{attribute 'global_init_slot' := '40510'}
VAR_GLOBAL
  LblAggregates_FunctionallyIndependentEequipment                 :FB_BA_Label:=( sObjName:='FIE',sDescr:='Functionally independent equipment');
  LblAggregates_SelfContainedControlUnit                          :FB_BA_Label:=( sObjName:='SCR',sDescr:='Self-contained control or regulation unit');
  LblAggregates_ControlCabinet                                    :FB_BA_Label:=( sObjName:='CCB',sDescr:='Control cabinet (trade-specific)');
//330 Doors, gates, windows, sun protection
  LblAggregates_WindowDrive                                       :FB_BA_Label:=( sObjName:='WIN',sDescr:='Window (drive)');
  LblAggregates_WindowContact                                     :FB_BA_Label:=( sObjName:='WIC',sDescr:='Window contact');
  LblAggregates_Blind                                             :FB_BA_Label:=( sObjName:='BLD',sDescr:='Blind');
  LblAggregates_Awning                                            :FB_BA_Label:=( sObjName:='AWN',sDescr:='Awning');
  LblAggregates_RollerShutters                                    :FB_BA_Label:=( sObjName:='ROS',sDescr:='Roller shutters');
  LblAggregates_Gate                                              :FB_BA_Label:=( sObjName:='GAT',sDescr:='Gate');
  LblAggregates_Door                                              :FB_BA_Label:=( sObjName:='DOR',sDescr:='Door');
  LblAggregates_DoorContact                                       :FB_BA_Label:=( sObjName:='DOC',sDescr:='Door contact');
  LblAggregates_Blackout                                          :FB_BA_Label:=( sObjName:='BLA',sDescr:='Blackout');
//412 Water plants
  LblAggregates_TraceHeating                                      :FB_BA_Label:=( sObjName:='THT',sDescr:='Trace heating');
  LblAggregates_ElectricHeating                                   :FB_BA_Label:=( sObjName:='EHT',sDescr:='Electric heating (warm water temperature preparation)');
  LblAggregates_WaterFilter                                       :FB_BA_Label:=( sObjName:='WFL',sDescr:='Water filter');
//421 Heat generation plants
  LblAggregates_Furnace                                           :FB_BA_Label:=( sObjName:='FUR',sDescr:='Furnace');
  LblAggregates_HeatExchanger                                     :FB_BA_Label:=( sObjName:='HEX',sDescr:='Heat exchanger');
//430 Ventilation and refrigeration systems
  LblAggregates_FanExhaustAir                                     :FB_BA_Label:=( sObjName:='EHF',sDescr:='Exhaust air fan');
  LblAggregates_Airwasher                                         :FB_BA_Label:=( sObjName:='AWA',sDescr:='Airwasher');
  LblAggregates_Humidifier                                        :FB_BA_Label:=( sObjName:='HUF',sDescr:='Humidifier');
  LblAggregates_HumidifierPump                                    :FB_BA_Label:=( sObjName:='HUP',sDescr:='Humidifier pump');
  LblAggregates_FireDamper                                        :FB_BA_Label:=( sObjName:='FID',sDescr:='Fire damper, fire protection valve');
  LblAggregates_SmokeProtectionDamper                             :FB_BA_Label:=( sObjName:='SPD',sDescr:='Smoke protection damper');
  LblAggregates_SmokeExtractorDamper                              :FB_BA_Label:=( sObjName:='SEP',sDescr:='Smoke extractor damper');
  LblAggregates_CeilingSwirlDiffuser                              :FB_BA_Label:=( sObjName:='CSD',sDescr:='Ceiling swirl diffuser');
  LblAggregates_RoofAirHeater                                     :FB_BA_Label:=( sObjName:='RAH',sDescr:='Roof air heater');
  LblAggregates_DirectEvaporator                                  :FB_BA_Label:=( sObjName:='DEA',sDescr:='Direct evaporator');
  LblAggregates_ElectricalAirHeater                               :FB_BA_Label:=( sObjName:='EAH',sDescr:='Electrical air heater');
  LblAggregates_ElectricReHeater                                  :FB_BA_Label:=( sObjName:='ERH',sDescr:='Electric re-heater');
  LblAggregates_ElectricaPreHeater                                :FB_BA_Label:=( sObjName:='EPH',sDescr:='Electrical pre-heater');
  LblAggregates_HeaterGeneral                                     :FB_BA_Label:=( sObjName:='HTR',sDescr:='Heater ');
  LblAggregates_FanExtractAir                                     :FB_BA_Label:=( sObjName:='EXF',sDescr:='Extract air fan ');
  LblAggregates_InductionDevice                                   :FB_BA_Label:=( sObjName:='IND',sDescr:='Induction device');
  LblAggregates_RefrigerantDryer                                  :FB_BA_Label:=( sObjName:='RFD',sDescr:='Refrigerant dryer');
  LblAggregates_CirculatorySystem                                 :FB_BA_Label:=( sObjName:='CCS',sDescr:='Circulatory system ');
  LblAggregates_AirFilterOutsideAir                               :FB_BA_Label:=( sObjName:='AFI',sDescr:='Outside air filter');
  LblAggregates_AirFilterSupplyAir                                :FB_BA_Label:=( sObjName:='AFI',sDescr:='Supply air filter');
  LblAggregates_AirFilterExhaustAir                               :FB_BA_Label:=( sObjName:='AFI',sDescr:='Exhaus air filter');
  LblAggregates_AirFilterExtractAir                               :FB_BA_Label:=( sObjName:='AFI',sDescr:='Extract air filter');
  LblAggregates_AirFilter                                         :FB_BA_Label:=( sObjName:='AFI',sDescr:='Air filter');
  LblAggregates_VentilationDamper                                 :FB_BA_Label:=( sObjName:='VFL',sDescr:='Ventilation flap');
  LblAggregates_VentilationDamperOutsideAir                       :FB_BA_Label:=( sObjName:='VFL',sDescr:='Ventilation flap outside air');
  LblAggregates_VentilationDamperExhaustAir                       :FB_BA_Label:=( sObjName:='VFL',sDescr:='Ventilation flap exhaust air');
  LblAggregates_VentilationDamperMixAir                           :FB_BA_Label:=( sObjName:='VFL',sDescr:='Ventilation flap mix air');
  LblAggregates_VentilationDamperSupplyAir                        :FB_BA_Label:=( sObjName:='VFL',sDescr:='Ventilation flap supply air');
  LblAggregates_VentilationDamperBypassAir                        :FB_BA_Label:=( sObjName:='VFL',sDescr:='Ventilation flap bypass');
  LblAggregates_Pump                                              :FB_BA_Label:=( sObjName:='PUM',sDescr:='Pump');
  LblAggregates_RecirculatingAirCoolingDevice                     :FB_BA_Label:=( sObjName:='RAC',sDescr:='Recirculating air cooling device');
  LblAggregates_FanRecirculatingAir                               :FB_BA_Label:=( sObjName:='RAF',sDescr:='Recirculating air fan');
  LblAggregates_UvFilter                                          :FB_BA_Label:=( sObjName:='UVF',sDescr:='UV filter');
  LblAggregates_VariableFlowRateController                        :FB_BA_Label:=( sObjName:='VFC',sDescr:='Variable flow rate controller');
  LblAggregates_WaterAirHeater                                    :FB_BA_Label:=( sObjName:='WAH',sDescr:='Water air heater');
  LblAggregates_WaterReHeater                                     :FB_BA_Label:=( sObjName:='WRH',sDescr:='Water re-heater');
  LblAggregates_WaterPreHeater                                    :FB_BA_Label:=( sObjName:='WPH',sDescr:='Water pre-heater');
  LblAggregates_HeatRecovery                                      :FB_BA_Label:=( sObjName:='HRC',sDescr:='Heat recovery');
  LblAggregates_FanSupplyAir                                      :FB_BA_Label:=( sObjName:='SUF',sDescr:='Supply air fan');
  LblAggregates_SmokeExtractionSystems                            :FB_BA_Label:=( sObjName:='SES',sDescr:='Smoke extraction systems');
  LblAggregates_SmokeExtractionVentilator                         :FB_BA_Label:=( sObjName:='SEF',sDescr:='Smoke extraction fan');
  LblAggregates_VentWindow                                        :FB_BA_Label:=( sObjName:='VWI',sDescr:='Vent window');
  LblAggregates_VentFlap                                          :FB_BA_Label:=( sObjName:='VFL',sDescr:='Vent flap');
  LblAggregates_VentDoor                                          :FB_BA_Label:=( sObjName:='VDO',sDescr:='Vent door');
  LblAggregates_WakeFan                                           :FB_BA_Label:=( sObjName:='WAF',sDescr:='Wake fan');
//434 Refrigeration systems
  LblAggregates_GlycoOilProtector                                 :FB_BA_Label:=( sObjName:='GLP',sDescr:='Glycol/oil protector');
  LblAggregates_Chiller                                           :FB_BA_Label:=( sObjName:='CHI',sDescr:='Chiller');
  LblAggregates_ReCoolingPlant                                    :FB_BA_Label:=( sObjName:='RCP',sDescr:='Re-cooling plant');
//440 High-voltage systems
  LblAggregates_GeneralPowerSupply                                :FB_BA_Label:=( sObjName:='GPS',sDescr:='General power supply');
  LblAggregates_CombindeHeatPowerStation                          :FB_BA_Label:=( sObjName:='CGU',sDescr:='Co-generation unit');
  LblAggregates_CompensationSystem                                :FB_BA_Label:=( sObjName:='CPS',sDescr:='Compensation system');
  LblAggregates_CouplingSwitch                                    :FB_BA_Label:=( sObjName:='COS',sDescr:='Coupling switch');
  LblAggregates_LoadBreakSwitch                                   :FB_BA_Label:=( sObjName:='LBS',sDescr:='Load-break switch');
  LblAggregates_CircuitBreaker                                    :FB_BA_Label:=( sObjName:='CCB',sDescr:='Circuit breaker');
  LblAggregates_NetworkAnalyser                                   :FB_BA_Label:=( sObjName:='NWA',sDescr:='Network analyser');
  LblAggregates_EmergencyPoweGeneratorUnit                        :FB_BA_Label:=( sObjName:='EPG',sDescr:='Emergency power generator unit');
  LblAggregates_EmergencyLighting                                 :FB_BA_Label:=( sObjName:='EML',sDescr:='Emergency lighting');
  LblAggregates_SafetyPowerSupply                                 :FB_BA_Label:=( sObjName:='SPS',sDescr:='Safety power supply');
  LblAggregates_Transformer                                       :FB_BA_Label:=( sObjName:='TRF',sDescr:='Transformer');
  LblAggregates_UninterruptiblePowerSupply                        :FB_BA_Label:=( sObjName:='UPS',sDescr:='Uninterruptible power supply');
//450 Telecommunications and information technology equipment
  LblAggregates_CentralFireAlarmSystem                            :FB_BA_Label:=( sObjName:='CFA',sDescr:='Central fire alarm system');
  LblAggregates_FireControlPanel                                  :FB_BA_Label:=( sObjName:='FCP',sDescr:='Fire control panel');
  LblAggregates_KitchenTableau                                    :FB_BA_Label:=( sObjName:='KIT',sDescr:='Kitchen tableau');
  LblAggregates_SmokeDetector                                     :FB_BA_Label:=( sObjName:='SDE',sDescr:='Smoke detector');
  LblAggregates_SmokeProtectionScreen                             :FB_BA_Label:=( sObjName:='SPS',sDescr:='Smoke protection screen');
  LblAggregates_VoiceAlarmCentre                                  :FB_BA_Label:=( sObjName:='VAC',sDescr:='Voice alarm centre');
  LblAggregates_Tableau                                           :FB_BA_Label:=( sObjName:='TAB',sDescr:='Tableau (general)');
//460 Conveyors
  LblAggregates_LiftGeneral                                       :FB_BA_Label:=( sObjName:='LIG',sDescr:='Lift general');
  LblAggregates_GoodsLift                                         :FB_BA_Label:=( sObjName:='GLI',sDescr:='Goods lift');
  LblAggregates_PassengerLift                                     :FB_BA_Label:=( sObjName:='PLI',sDescr:='Passenger lift');
//470 User-specific systems
  LblAggregates_FumeCupboard                                      :FB_BA_Label:=( sObjName:='FCB',sDescr:='Fume cupboard');
  LblAggregates_Compressor                                        :FB_BA_Label:=( sObjName:='COM',sDescr:='Compressor');
  LblAggregates_ProgrammableLogicControllers                      :FB_BA_Label:=( sObjName:='PLC',sDescr:='Programmable logic controllers');
//479 User-specific system, weather station
  LblAggregates_RainSensor                                        :FB_BA_Label:=( sObjName:='RAS',sDescr:='Rain sensor');
  LblAggregates_SolarRadiation                                    :FB_BA_Label:=( sObjName:='SOR',sDescr:='Solar radiation');
  LblAggregates_WeatherStation                                    :FB_BA_Label:=( sObjName:='WST',sDescr:='Weather station');
  LblAggregates_WindSpeed                                         :FB_BA_Label:=( sObjName:='WIS',sDescr:='Wind speed');
  LblAggregates_WindDirection                                     :FB_BA_Label:=( sObjName:='WID',sDescr:='Wind direction');
  LblAggregates_WindForce                                         :FB_BA_Label:=( sObjName:='WDF',sDescr:='Wind force');
  LblAggregates_Brightness                                        :FB_BA_Label:=( sObjName:='BIN',sDescr:='Brightness');
  LblAggregates_Dawn                                              :FB_BA_Label:=( sObjName:='BID',sDescr:='Brightness dawn');
  LblAggregates_PressureAbsolute                                  :FB_BA_Label:=( sObjName:='PAB',sDescr:='Pressure absolute');
  LblAggregates_PressureRelative                                  :FB_BA_Label:=( sObjName:='PRE',sDescr:='Pressure relative');
  LblAggregates_GeoLatitude                                       :FB_BA_Label:=( sObjName:='LAT',sDescr:='Latitude       ');
  LblAggregates_GeoLongitude                                      :FB_BA_Label:=( sObjName:='LOT',sDescr:='Longitude      ');
  LblAggregates_SunAzimuth                                        :FB_BA_Label:=( sObjName:='AZI',sDescr:='Azimuth        ');
  LblAggregates_SunElevation                                      :FB_BA_Label:=( sObjName:='ELE',sDescr:='Elevation      ');
//480 Building automation and control systems
  LblAggregates_SystemSwitch                                      :FB_BA_Label:=( sObjName:='SYS',sDescr:='System switch');
  LblAggregates_AutomationStationEquipment                        :FB_BA_Label:=( sObjName:='ASE',sDescr:='Automation station equipment');
  LblAggregates_BusLineCoupler                                    :FB_BA_Label:=( sObjName:='BUS',sDescr:='Bus line coupler');
  LblAggregates_DataInterfaceUnit                                 :FB_BA_Label:=( sObjName:='DIU',sDescr:='Data interface unit');
  LblAggregates_FieldbusModule                                    :FB_BA_Label:=( sObjName:='FBM',sDescr:='Fieldbus module');
  LblAggregates_InformationFocalPoint                             :FB_BA_Label:=( sObjName:='IFP',sDescr:='Information focal point');
  LblAggregates_ManagementAndControlEquipment                     :FB_BA_Label:=( sObjName:='MCE',sDescr:='Management and control equipment');
//481 BACS sensors – temperature
  LblAggregates_TemperatureGasEmission                            :FB_BA_Label:=( sObjName:='TEG',sDescr:='Emissions gas temperature');
  LblAggregates_TemperatureExtractAir                             :FB_BA_Label:=( sObjName:='TEX',sDescr:='Extract air temperature');
  LblAggregates_TemperatureOutside                                :FB_BA_Label:=( sObjName:='TOU',sDescr:='Outside temperature');
  LblAggregates_TemperatureExhaustAir                             :FB_BA_Label:=( sObjName:='TEH',sDescr:='Exhaust air temperature');
  LblAggregates_FrostProtectionMonitor                            :FB_BA_Label:=( sObjName:='FPM',sDescr:='Frost protection monitor');
  LblAggregates_TemperatureMixedAir                               :FB_BA_Label:=( sObjName:='TMI',sDescr:='Mixed air temperature');
  LblAggregates_TemperatureRoomAir                                :FB_BA_Label:=( sObjName:='TRO',sDescr:='Room temperature');
  LblAggregates_TemperatureReturnFlow                             :FB_BA_Label:=( sObjName:='TRT',sDescr:='Return flow temperature');
  LblAggregates_LimiterSafetyTemperature                          :FB_BA_Label:=( sObjName:='STL',sDescr:='Safety temperature limiter');
  LblAggregates_MonitorSafetyTemperature                          :FB_BA_Label:=( sObjName:='STM',sDescr:='Safety temperature monitor');
  LblAggregates_TemperatureStorage                                :FB_BA_Label:=( sObjName:='TST',sDescr:='Storage temperature');
  LblAggregates_TemperatureDewPoint                               :FB_BA_Label:=( sObjName:='TDP',sDescr:='Dew point temperature');
  LblAggregates_MonitorDewPoint                                   :FB_BA_Label:=( sObjName:='DPM',sDescr:='Dew point monitor');
  LblAggregates_TemperatureAfterCooler                            :FB_BA_Label:=( sObjName:='TAC',sDescr:='Temperature after cooler');
  LblAggregates_TemperatureAfterPreHeater                         :FB_BA_Label:=( sObjName:='TAP',sDescr:='Temperature after pre-heater');
  LblAggregates_TemperatureAfterHeatRecovery                      :FB_BA_Label:=( sObjName:='TAR',sDescr:='Temperature after heat recovery');
  LblAggregates_Thermostat                                        :FB_BA_Label:=( sObjName:='THM',sDescr:='Thermostat');
  LblAggregates_TemperatureHotWater                               :FB_BA_Label:=( sObjName:='THW',sDescr:='Hot water temperature');
  LblAggregates_TemperatureCirculation                            :FB_BA_Label:=( sObjName:='TCI',sDescr:='Circulation temperature');
  LblAggregates_TemperatureRecirculatingAir                       :FB_BA_Label:=( sObjName:='TRE',sDescr:='Recirculating air temperature');
  LblAggregates_TemperatureFlow                                   :FB_BA_Label:=( sObjName:='TFL',sDescr:='Flow temperature');
  LblAggregates_TemperatureSupplyAir                              :FB_BA_Label:=( sObjName:='TSU',sDescr:='Supply air temperature');
//481 BACS sensors – pressure
  LblAggregates_PressureExtractAir                                :FB_BA_Label:=( sObjName:='PEX',sDescr:='Extract air pressure');
  LblAggregates_PressureOutsideAir                                :FB_BA_Label:=( sObjName:='POU',sDescr:='Outside air pressure');
  LblAggregates_PressureDifferential                              :FB_BA_Label:=( sObjName:='PDI',sDescr:='Differential pressure');
  LblAggregates_PressureDifferentialOutsideAirFilter              :FB_BA_Label:=( sObjName:='PDI',sDescr:='Differential pressure outside air filter');
  LblAggregates_PressureDifferentialExtractAirFilter              :FB_BA_Label:=( sObjName:='PDI',sDescr:='Differential pressure extract air filter');
  LblAggregates_PressureDifferentialExhaustAirFilter              :FB_BA_Label:=( sObjName:='PDI',sDescr:='Differential pressure exhaust air filter');
  LblAggregates_PressureDifferentialSupplyAirFan                  :FB_BA_Label:=( sObjName:='PDI',sDescr:='Differential pressure supply air fan');
  LblAggregates_PressureDifferentialExtractAirFan                 :FB_BA_Label:=( sObjName:='PDI',sDescr:='Differential pressure ectract air fan');
  LblAggregates_PressureDifferentialExhaustAirFan                 :FB_BA_Label:=( sObjName:='PDI',sDescr:='Differential pressure exhaust air fan');
  LblAggregates_PressureSensorFlow                                :FB_BA_Label:=( sObjName:='PFL',sDescr:='Pressure sensor (water) flow');
  LblAggregates_MonitorPressure                                   :FB_BA_Label:=( sObjName:='PCO',sDescr:='Pressure controller');
  LblAggregates_PressureExhaustAir                                :FB_BA_Label:=( sObjName:='PEH',sDescr:='Exhaust air pressure');
  LblAggregates_PressureRoomAir                                   :FB_BA_Label:=( sObjName:='PRO',sDescr:='Room pressure');
  LblAggregates_PressureIndexCircuitSensorDifferential            :FB_BA_Label:=( sObjName:='PSI',sDescr:='Index circuit sensor differential pressure');
  LblAggregates_LimiterSafetyPressure                             :FB_BA_Label:=( sObjName:='SPL',sDescr:='Safety pressure limiter');
  LblAggregates_PressureSupplyAir                                 :FB_BA_Label:=( sObjName:='PSU',sDescr:='Supply air pressure');
//481 BACS sensors – air quality
  LblAggregates_CO2Sensor                                         :FB_BA_Label:=( sObjName:='COM',sDescr:='CO2 sensor');
  LblAggregates_QualityExtractAir                                 :FB_BA_Label:=( sObjName:='QEX',sDescr:='Extract air quality');
  LblAggregates_OualityRoomAir                                    :FB_BA_Label:=( sObjName:='QRO',sDescr:='Room air quality');
  LblAggregates_QualitiySupplyAir                                 :FB_BA_Label:=( sObjName:='QSU',sDescr:='Supply air quality');
  LblAggregates_QualityAirSensor                                  :FB_BA_Label:=( sObjName:='AQS',sDescr:='Air quality sensor');
//481 BACS sensors – humidity
  LblAggregates_Hygrostat                                         :FB_BA_Label:=( sObjName:='HYG',sDescr:='Hygrostat');
  LblAggregates_RelativeHumiditiyExtractAir                       :FB_BA_Label:=( sObjName:='HEX',sDescr:='Relative extract air humidity');
  LblAggregates_RelativeHumidityOutsideAir                        :FB_BA_Label:=( sObjName:='HOU',sDescr:='Relative outside air humidity');
  LblAggregates_RelativeHumidityExhaustAir                        :FB_BA_Label:=( sObjName:='HEH',sDescr:='Relative exhaust air humidity');
  LblAggregates_MonitorCondensation                               :FB_BA_Label:=( sObjName:='HCM',sDescr:='Condensation monitor');
  LblAggregates_RelativeHumidityMixedAir                          :FB_BA_Label:=( sObjName:='HMI',sDescr:='Relative mixed air humidity');
  LblAggregates_RelativeHumidityRoomHumidity                      :FB_BA_Label:=( sObjName:='HRO',sDescr:='Relative room humidity');
  LblAggregates_RelativeHumidityRecirculatedAir                   :FB_BA_Label:=( sObjName:='HRE',sDescr:='Relative recirculated air humidity');
  LblAggregates_RelativeHumiditySupplyAir                         :FB_BA_Label:=( sObjName:='HSU',sDescr:='Relative supply air humidity');
  LblAggregates_AbsoluteHumidityExtractAir                        :FB_BA_Label:=( sObjName:='XEX',sDescr:='Absolute extract air humidity');
  LblAggregates_AbsoluteHumidtiyOutsideAir                        :FB_BA_Label:=( sObjName:='XOU',sDescr:='Absolute outsie air humidity');
  LblAggregates_AbsoluteHumidtiyExhaustAir                        :FB_BA_Label:=( sObjName:='XEH',sDescr:='Absolute exhaust air humidity');
  LblAggregates_AbsoluteHumidityMixedAir                          :FB_BA_Label:=( sObjName:='XMI',sDescr:='Absolute mixed air humidity');
  LblAggregates_AbsoluteHumidityRoomAir                           :FB_BA_Label:=( sObjName:='XRO',sDescr:='Absolute room humidity');
  LblAggregates_AbsoluteHumidityRecirculatingAir                  :FB_BA_Label:=( sObjName:='XRE',sDescr:='Absolute recirculating air humidity');
  LblAggregates_AbsoluteHumiditySupplyAir                         :FB_BA_Label:=( sObjName:='XSU',sDescr:='Absolute supply air humidity');
//481 BACS sensors – consumption recording
  LblAggregates_MeterElectric                                     :FB_BA_Label:=( sObjName:='ELM',sDescr:='Electric meter');
  LblAggregates_MeterGasNaturalGas                                :FB_BA_Label:=( sObjName:='GAM',sDescr:='Gas meter natural gas');
  LblAggregates_MeterCoolingEnergy                                :FB_BA_Label:=( sObjName:='CEM',sDescr:='Cooling energy meter');
  LblAggregates_MeterHeat                                         :FB_BA_Label:=( sObjName:='HEM',sDescr:='Heat meter');
  LblAggregates_MetferWater                                       :FB_BA_Label:=( sObjName:='WAM',sDescr:='Water meter');
  LblAggregates_MeterFuel                                         :FB_BA_Label:=( sObjName:='FUM',sDescr:='Fuel meter (oil)');
  LblAggregates_MeterSteam                                        :FB_BA_Label:=( sObjName:='STM',sDescr:='Steam meter');
  LblAggregates_DegreeDayNumber                                   :FB_BA_Label:=( sObjName:='DDN',sDescr:='Degree day number');
//481 BACS sensors – condition recording and other
  LblAggregates_LeakageMonitoring                                 :FB_BA_Label:=( sObjName:='LKM',sDescr:='Leakage monitoring');
  LblAggregates_EmergencyStop                                     :FB_BA_Label:=( sObjName:='EMG',sDescr:='Emergency stop unit/button');
  LblAggregates_StockLevel                                        :FB_BA_Label:=( sObjName:='SLV',sDescr:='Stock level');
  LblAggregates_FlowMonitor                                       :FB_BA_Label:=( sObjName:='FLM',sDescr:='Flow monitor');
  LblAggregates_OverflowMonitoring                                :FB_BA_Label:=( sObjName:='OVM',sDescr:='Overflow monitoring');
  LblAggregates_LowWaterCutOff                                    :FB_BA_Label:=( sObjName:='WCO',sDescr:='Low-water cut-off');
  LblAggregates_WaterFlowMonitor                                  :FB_BA_Label:=( sObjName:='WFM',sDescr:='Water flow monitor');
//481 BACS sensors – speed
  LblAggregates_PumpSpeed                                         :FB_BA_Label:=( sObjName:='SPU',sDescr:='Pump speed');
  LblAggregates_FanSpeedExtractAir                                :FB_BA_Label:=( sObjName:='SEX',sDescr:='Fan speed (extract air)');
  LblAggregates_FanSpeedExhaustAir                                :FB_BA_Label:=( sObjName:='SEH',sDescr:='Fan speed (exhaust air)');
  LblAggregates_FanSpeedSupplyAir                                 :FB_BA_Label:=( sObjName:='SSU',sDescr:='Fan speed (supply air)');
//481 BACS sensors – volume flow
  LblAggregates_VolumeFlowRateExtractAir                          :FB_BA_Label:=( sObjName:='VEX',sDescr:='Extract air volume flow rate');
  LblAggregates_VolumeFlowRateOutsideAir                          :FB_BA_Label:=( sObjName:='VOU',sDescr:='Outside air volume flow rate');
  LblAggregates_VolumeFlowRateExhaustAir                          :FB_BA_Label:=( sObjName:='VEH',sDescr:='Exhaust air volume flow rate');
  LblAggregates_VolumeFlowRateBrineCirculatorySystem              :FB_BA_Label:=( sObjName:='VBR',sDescr:='Volume flow brine (circulatory system)');
  LblAggregates_VolumeFlowRateColdDrinkingWater                   :FB_BA_Label:=( sObjName:='VCW',sDescr:='Volume flow cold drinking water');
  LblAggregates_VolumeFlowRateHotDrinkingWater                    :FB_BA_Label:=( sObjName:='VHW',sDescr:='Volume flow hot drinking water');
  LblAggregates_VolumeFlowRateWaterPurification                   :FB_BA_Label:=( sObjName:='VWP',sDescr:='Volume flow water purification');
  LblAggregates_VolumeFlowRateSupplyAir                           :FB_BA_Label:=( sObjName:='VSU',sDescr:='Supply air volume flow');
//481 BACS actuators – actuating drives
  LblAggregates_ValveRadiator                                     :FB_BA_Label:=( sObjName:='RDV',sDescr:='Radiator valve drive');
  LblAggregates_ValveCoolingCeiling                               :FB_BA_Label:=( sObjName:='CCV',sDescr:='Cooling ceiling valve drive');
  LblAggregates_MotorisedFlap                                     :FB_BA_Label:=( sObjName:='FLA',sDescr:='Motorised flap');
  LblAggregates_Valve                                             :FB_BA_Label:=( sObjName:='VLV',sDescr:='Motor valve');
  LblAggregates_HumidifierValve                                   :FB_BA_Label:=( sObjName:='VLV',sDescr:='Humidifier valve');
//481 BACS lighting
  LblAggregates_IlluminationExternal                              :FB_BA_Label:=( sObjName:='EOU',sDescr:='Illumination outside');
  LblAggregates_IlluminationRoom                                  :FB_BA_Label:=( sObjName:='ERO',sDescr:='Illumination room');
  LblAggregates_LightColourRoom                                   :FB_BA_Label:=( sObjName:='CRO',sDescr:='Light colour room');
  LblAggregates_RedLightIntensity                                 :FB_BA_Label:=( sObjName:='LRD',sDescr:='Red light intensity');
  LblAggregates_GreenLightIntensity                               :FB_BA_Label:=( sObjName:='LGN',sDescr:='Green light intensity');
  LblAggregates_BlueLightIntensity                                :FB_BA_Label:=( sObjName:='LBL',sDescr:='Blue light intensity');
//481 BACS sun protection
  LblAggregates_BlindAnglePosition                                :FB_BA_Label:=( sObjName:='BAP',sDescr:='Blind angle position');
  LblAggregates_ShadingPosition                                   :FB_BA_Label:=( sObjName:='BSP',sDescr:='Shading position');
  LblAggregates_MovementCommand                                   :FB_BA_Label:=( sObjName:='BMC',sDescr:='Blind Movement command');
//485 Room automation
  LblAggregates_DisplayAndControlUnit                             :FB_BA_Label:=( sObjName:='DCU',sDescr:='Display and control unit');
  LblAggregates_PresenceSwitches                                  :FB_BA_Label:=( sObjName:='PDE',sDescr:='Presence switches, detectors, motion detectors');
  LblAggregates_RoomAutomationDevice                              :FB_BA_Label:=( sObjName:='RAD',sDescr:='Room automation device');
  LblAggregates_RoomControlUnit                                   :FB_BA_Label:=( sObjName:='RCU',sDescr:='Room control unit');
END_VAR

// ---- Templates/GVLs/DPAD/Labels/1033/LblControl1033.TcGVL
{region '#Template'}
	{attribute 'Version' := '1.0.0.0'}
	{attribute 'Tags' := '"LCID": "1031", "Text": "GVL, AKS, Labels, ObjectName, Description"'}
	{attribute 'Tags' := '"LCID": "1033", "Text": "GVL, DPAD, Labels, ObjectName, Description"'}
	{attribute 'Description' := '"LCID": "1031", "Text": "Anlagenkennzeichnungssystem, Labels controls"'}
	{attribute 'Description' := '"LCID": "1033", "Text": "Data Point Addressing Description, Labels controls"'}
{endregion}
	 
{attribute 'global_init_slot' := '40510'}
VAR_GLOBAL
  LblControl_OperationMode                                     :FB_BA_Label:=( sObjName:='OPM',sDescr:='Operation Mode');
  LblControl_SummerNightCooling                                :FB_BA_Label:=( sObjName:='SNC',sDescr:='Summer night cooling');
  LblControl_DifferencePressureMonitoringSupplyAirFan          :FB_BA_Label:=( sObjName:='DPM',sDescr:='Difference Pressure Monitoring Supply Air Fan');
  LblControl_DifferencePressureMonitoringExtractAirFan         :FB_BA_Label:=( sObjName:='DPM',sDescr:='Difference Pressure Monitoring Extract Air Fan');
  LblControl_TSetpointCalculation                              :FB_BA_Label:=( sObjName:='SPC',sDescr:='Setpoint Calculation Temperature');
  LblControl_HSetpointCalculation                              :FB_BA_Label:=( sObjName:='SPC',sDescr:='Setpoint Calculation Humidity');
  LblControl_TCascadeSupplyAirControl                          :FB_BA_Label:=( sObjName:='CTL',sDescr:='Cascade control supply air temperature');
  LblControl_HCascadeSupplyAirControl                          :FB_BA_Label:=( sObjName:='CTL',sDescr:='Cascade control supply air humidity');
  LblControl_PreHeater                                         :FB_BA_Label:=( sObjName:='PRH',sDescr:='PreHeater');
  LblControl_ReHeater                                          :FB_BA_Label:=( sObjName:='RHE',sDescr:='Reheater');
  LblControl_EnergyRecovery                                    :FB_BA_Label:=( sObjName:='ERC',sDescr:='Energy Recovery');
  LblControl_SupplyAirTemperatureControl                       :FB_BA_Label:=( sObjName:='CTL',sDescr:='Supply Air Temperature Control');
  LblControl_SupplyAirDehumidifierControl                      :FB_BA_Label:=( sObjName:='CTL',sDescr:='Supply Air Dehumidification Control');
  LblControl_SupplyAirHumidifierController                     :FB_BA_Label:=( sObjName:='CTL',sDescr:='Supply Air Humidity Control');
  LblControl_SupplyAirTemperatureLimitationControl             :FB_BA_Label:=( sObjName:='CTL',sDescr:='Supply Air Temperature Limitation Control');
  LblControl_ReturnWaterControl                                :FB_BA_Label:=( sObjName:='CTL',sDescr:='Return Water Control');
  LblControl_HumidityLimitationControl                         :FB_BA_Label:=( sObjName:='CTL',sDescr:='Rel humidity limitation control');
  LblControl_CalculationPreRinseSetpoint                       :FB_BA_Label:=( sObjName:='SPC',sDescr:='Calculation PreRinse Setpoint');
  LblControl_FrostProtectionControl                            :FB_BA_Label:=( sObjName:='FPC',sDescr:='Frost Protection Control');
  LblControl_ExhaustAirTemperatureControl                      :FB_BA_Label:=( sObjName:='CTL',sDescr:='Exhaust Air Temperature Control');
  LblControl_EnergyRecoveryDeicingRamp                         :FB_BA_Label:=( sObjName:='RMP',sDescr:='Energy Recovery Deicing Ramp');
  LblControl_BACnetDevice                                      :FB_BA_Label:=( sObjName:='DEV',sDescr:='BACnet device');
  LblControl_PlantControl                                      :FB_BA_Label:=( sObjName:='PCT',sDescr:='Plant Control');
  LblControl_TSequenceControl                                  :FB_BA_Label:=( sObjName:='SEQ',sDescr:='Sequence Control Temp');
  LblControl_HSequenceControl                                  :FB_BA_Label:=( sObjName:='SEQ',sDescr:='Sequence Control Humidity');
  LblControl_GeneralBeckhoffEventClass                         :FB_BA_Label:=( sObjName:='ECL',sDescr:='Event class');
  LblControl_GeneralSettings                                   :FB_BA_Label:=( sObjName:='SYP',sDescr:='System parameters');
  LblControl_GeneralCabinetBasicEquipment                      :FB_BA_Label:=( sObjName:='CBE',sDescr:='Cabinet basic equipment');
  LblControl_GeneralCabinetAdditionalEquipment                 :FB_BA_Label:=( sObjName:='CAE',sDescr:='Cabinet additional equipment');
  LblControl_EventIndicationLamp                               :FB_BA_Label:=( sObjName:='CEM',sDescr:='Collective error message lamp');
  LblControl_AcknowledgeCommand                                :FB_BA_Label:=( sObjName:='ACK',sDescr:='Acknowledge Hardware');
  LblControl_RemoteAcknowledgement                             :FB_BA_Label:=( sObjName:='ACK',sDescr:='Remote acknowledgement fault');
  LblControl_LocalAcknowledgement                              :FB_BA_Label:=( sObjName:='ACK',sDescr:='Local acknowledgement fault');
  LblControl_Acknowledge                                       :FB_BA_Label:=( sObjName:='ACK',sDescr:='Acknowledge');
// 
  LblControl_Fuse                                              :FB_BA_Label:=( sObjName:='FUS',sDescr:='Fuse');
// Settings
  LblControl_FrostProtection                                   :FB_BA_Label:=( sObjName:='FRP',sDescr:='Frost protection');
  LblControl_MinimumOutsideTemperature                         :FB_BA_Label:=( sObjName:='TWT',sDescr:='Minimum outdoor temperature');
  LblControl_TemperatureWeatherLowLimit                        :FB_BA_Label:=( sObjName:='TWT',sDescr:='Temperature weather low limit');
  LblControl_TemperatureWeatherDamped                          :FB_BA_Label:=( sObjName:='TWD',sDescr:='Temperature weather damped');
  LblControl_TemperatureWeatherDampedLowLimit                  :FB_BA_Label:=( sObjName:='TWD',sDescr:='Temperature Weather damped low limit');
  LblControl_PressureControl                                   :FB_BA_Label:=( sObjName:='CTL',sDescr:='Pressure control');
  LblControl_Converter3Point                                   :FB_BA_Label:=( sObjName:='CNV',sDescr:='3 point converter');
  LblControl_HeatingCurve                                      :FB_BA_Label:=( sObjName:='HCV',sDescr:='Heating curve');
  LblControl_SetpointGeneration                                :FB_BA_Label:=( sObjName:='SPG',sDescr:='Setpoint generation');
  LblControl_RequestHeatState                                  :FB_BA_Label:=( sObjName:='RHS',sDescr:='Request heat state');
  LblControl_RequestHeatSetpoint                               :FB_BA_Label:=( sObjName:='RHS',sDescr:='Request heat setpoint');
  LblControl_FlowTempControl                                   :FB_BA_Label:=( sObjName:='CTL',sDescr:='Flow temperature control');
// 
  LblControl_RoomTemperatureControl                            :FB_BA_Label:=( sObjName:='RGL',sDescr:='Room Temperature Control');
  LblControl_FlowTemperatureControl                            :FB_BA_Label:=( sObjName:='CTL',sDescr:='Flow temperature control');
  LblControl_SetpointHeating                                   :FB_BA_Label:=( sObjName:='SPG',sDescr:='Setpoint generation heating');
  LblControl_SetpointCooling                                   :FB_BA_Label:=( sObjName:='SPG',sDescr:='Setpoint generation cooling');
  LblControl_Facade                                            :FB_BA_Label:=( sObjName:='FIE',sDescr:='Facade Data');
  LblControl_BuildingAlarms                                    :FB_BA_Label:=( sObjName:='FIE',sDescr:='Building Alarms');
  LblControl_BuildingEnergyLevel                               :FB_BA_Label:=( sObjName:='FIE',sDescr:='Building Energylevel');
  LblControl_BuildingMode                                      :FB_BA_Label:=( sObjName:='FIE',sDescr:='Building Operationmode');
  LblControl_BuildingSpRmT                                     :FB_BA_Label:=( sObjName:='FIE',sDescr:='Building Roomtemperature Setpoints');
  LblControl_BuildingSunprotection                             :FB_BA_Label:=( sObjName:='FIE',sDescr:='Building Sunprotection');
  LblControl_TemperatureFrost                                  :FB_BA_Label:=( sObjName:='TFR',sDescr:='Temperature Frost');
  LblControl_MixedAirStartUpRamp                               :FB_BA_Label:=( sObjName:='RMP',sDescr:='Ramp plant start');
  LblControl_Cooler                                            :FB_BA_Label:=( sObjName:='COL',sDescr:='Cooler');
  LblControl_EvtCategoryLifeSafty                              :FB_BA_Label:=( sObjName:='ECL',sDescr:='Life safety');
  LblControl_EvtCategoryAlarmTechnical                         :FB_BA_Label:=( sObjName:='ECT',sDescr:='Technical alarm');
  LblControl_EvtCategoryDisturbance                            :FB_BA_Label:=( sObjName:='ECD',sDescr:='Disturbance');
  LblControl_EvtCategoryMaintenance                            :FB_BA_Label:=( sObjName:='ECM',sDescr:='Maintenance');
  LblControl_EvtCategoryNotification                           :FB_BA_Label:=( sObjName:='ECN',sDescr:='Notification');
  LblControl_EvtCategoryOther                                  :FB_BA_Label:=( sObjName:='ECO',sDescr:='Other');
  LblControl_TrendLogging                                      :FB_BA_Label:=( sObjName:='TRL',sDescr:='TrendLogging                                      ');
  LblControl_WeatherParameters                                 :FB_BA_Label:=( sObjName:='WTP',sDescr:='Weather Parameters');
  LblControl_SetpointFrostProtection                           :FB_BA_Label:=( sObjName:='SP_',sDescr:='Setpoint frost protection');
  LblControl_SetpointWeatherIcing                              :FB_BA_Label:=( sObjName:='SP_',sDescr:='Setpoint icing');
  LblControl_SetpointMinimumOutsideTemperature                 :FB_BA_Label:=( sObjName:='SPI',sDescr:='Setpoint minimum outside temperature');
  LblControl_MeanDamped                                        :FB_BA_Label:=( sObjName:='MWD',sDescr:='Mean value weather temperature damped');
  LblControl_OperationalMessageTemperatureWeatherLowLimit      :FB_BA_Label:=( sObjName:='OM_',sDescr:='Operational Message Temperature Weather Low Limit');
  LblControl_OperationalMessageTemperatureWeatherDampedLowLimit:FB_BA_Label:=( sObjName:='OM_',sDescr:='Operational Message Temperature Weather Damped Low Limit');
// Beckhoff Cabinet basic equipment
  LblControl_SwitchingCommandCollectiveFaultSignalLamp         :FB_BA_Label:=( sObjName:='SC_',sDescr:='Collective fault signal lamp switching command');
  LblControl_SwitchingCommandHardwareAcknowledgement           :FB_BA_Label:=( sObjName:='SC_',sDescr:='Hardware acknowledgement switching command');
  LblControl_ButtonRemoteAcknowledgement                       :FB_BA_Label:=( sObjName:='BUT',sDescr:='Input remote acknowledgement');
  LblControl_ButtonLocalAcknowledgement                        :FB_BA_Label:=( sObjName:='BUT',sDescr:='Button acknowledgement');
// Beckhoff Heating Circuit
  LblControl_HeatingLimit                                      :FB_BA_Label:=( sObjName:='HLM',sDescr:='Heating limit ');
  LblControl_PresentOperationMode                              :FB_BA_Label:=( sObjName:='POM',sDescr:='Present operation mode');
  LblControl_OperationModeSelection                            :FB_BA_Label:=( sObjName:='OMS',sDescr:='Operation mode selection');
// Beckhoff Summer Night Cooling
  LblControl_HysteresisRoomTemperature                         :FB_BA_Label:=( sObjName:='HYS',sDescr:='Hyeresis room temperature');
  LblControl_OutsideTemperatureLowLimit                        :FB_BA_Label:=( sObjName:='MIN',sDescr:='minimum outside temperature');
  LblControl_OffValueDifferenceOutsideInsightTemperature       :FB_BA_Label:=( sObjName:='MIN',sDescr:='Off Value differenz between ouside and insight temperature');
  LblControl_OnValueDifferenceOutsideInsightTemperature        :FB_BA_Label:=( sObjName:='MAX',sDescr:='On Value differenz between ouside and insight temperature');
// Beckhoff Damper
  LblControl_DriveTimeOpen                                     :FB_BA_Label:=( sObjName:='DTO',sDescr:='Drive time open');
  LblControl_DriveTimeClose                                    :FB_BA_Label:=( sObjName:='DTC',sDescr:='Drive time close');
  LblControl_DisturbanceFeedbackOpen                           :FB_BA_Label:=( sObjName:='DSO',sDescr:='Disturbance_feedback_open');
  LblControl_DisturbanceFeedbackClose                          :FB_BA_Label:=( sObjName:='DSC',sDescr:='Disturbance_feedback_close');
// 
  LblControl_TimeDelay                                         :FB_BA_Label:=( sObjName:='TD_',sDescr:='Time delay ');
  LblControl_TimeDelayFeedback                                 :FB_BA_Label:=( sObjName:='TDF',sDescr:='Time delay feedback');
  LblControl_TimeDelayInterruptionFeedback                     :FB_BA_Label:=( sObjName:='TDI',sDescr:='Time delay interruption');
// Beckhoff pre rins
  LblControl_PreRinseDuration                                  :FB_BA_Label:=( sObjName:='PRD',sDescr:='Pre rins duration');
  LblControl_DisturbancePreRinse                               :FB_BA_Label:=( sObjName:='DST',sDescr:='Disturbance pre rinse');
  LblControl_SetpointMinimalReturnWaterTemperature             :FB_BA_Label:=( sObjName:='SP_',sDescr:='Setpoint minimal return water temperature');
// Beckhoff ramp 
  LblControl_RampTimeUp                                        :FB_BA_Label:=( sObjName:='RTU',sDescr:='Ramp time up');
  LblControl_RampTimeDown                                      :FB_BA_Label:=( sObjName:='RTD',sDescr:='Ramp time down');
  LblControl_CommandOpen                                       :FB_BA_Label:=( sObjName:='SC_',sDescr:='Switch command open');
  LblControl_CommandClose                                      :FB_BA_Label:=( sObjName:='SC_',sDescr:='Switch command close');
  LblControl_CalculatedValue                                   :FB_BA_Label:=( sObjName:='CAV',sDescr:='calculated value');
  LblControl_Value                                             :FB_BA_Label:=( sObjName:='VAL',sDescr:='Value');
// Beckhoff event class
  LblControl_EvtClassSimple                                    :FB_BA_Label:=( sObjName:='NC_',sDescr:='Simple');
  LblControl_EvtClassStandard                                  :FB_BA_Label:=( sObjName:='NC_',sDescr:='Standard');
  LblControl_EvtClassExtended                                  :FB_BA_Label:=( sObjName:='NC_',sDescr:='Extended');
  LblControl_FlowSwitch                                        :FB_BA_Label:=( sObjName:='OM_',sDescr:='Operating message flow monitor');
  LblControl_SmokeAlarm                                        :FB_BA_Label:=( sObjName:='DST',sDescr:='Disturbance smoke alarm');
  LblControl_SystemFailure                                     :FB_BA_Label:=( sObjName:='DST',sDescr:='Disturbance system failure');
  LblControl_Contamination                                     :FB_BA_Label:=( sObjName:='DST',sDescr:='Disturbance Contamination');
  LblControl_SwitchingCommandSmokeDetector                     :FB_BA_Label:=( sObjName:='SC_',sDescr:='Switching command acknowledge');
  LblControl_ButtonReset                                       :FB_BA_Label:=( sObjName:='BUT',sDescr:='Button acknowledge');
  LblControl_OffsetNightSetpoint                               :FB_BA_Label:=( sObjName:='ONS',sDescr:='Offset night setback');
// 
  LblControl_SetpointRelHumidityHumidification                 :FB_BA_Label:=( sObjName:='SP_',sDescr:='Setpoint Relative Humidity Humidification');
  LblControl_SetpointRelHumidityDehumidification               :FB_BA_Label:=( sObjName:='SP_',sDescr:='Setpoint Relative Humidity Dehumidification');
  LblControl_SetpointAbsHumidityHumidification                 :FB_BA_Label:=( sObjName:='SPC',sDescr:='Setpoint absolute humidity humidification');
  LblControl_SetpointAbsHumidityDehumidification               :FB_BA_Label:=( sObjName:='SPC',sDescr:='Setpoint absolute humidity dehumidification');
  LblControl_SetpointRelHumidity                               :FB_BA_Label:=( sObjName:='SP_',sDescr:='Setpoint relative humidity');
  LblControl_SetpointAbsHumidity                               :FB_BA_Label:=( sObjName:='SP_',sDescr:='Setpoint absolute humidity');
  LblControl_OperationalMessageDehumidification                :FB_BA_Label:=( sObjName:='OM_',sDescr:='Operational message dehumidification');
// 
  LblControl_SetpointSunblindPosition                          :FB_BA_Label:=( sObjName:='SP_',sDescr:='Setpoint blind position');
  LblControl_SetpointSunblindAngle                             :FB_BA_Label:=( sObjName:='SP_',sDescr:='Setpoint blind angle');
  LblControl_CommandSunblindStart                              :FB_BA_Label:=( sObjName:='SC_',sDescr:='Command sunblind start');
  LblControl_ButtonSunblind                                    :FB_BA_Label:=( sObjName:='BUT',sDescr:='Sun blind button');
  LblControl_FeedbackSunblindPosition                          :FB_BA_Label:=( sObjName:='FDB',sDescr:='Feedback blind position');
  LblControl_FeedbackSunblindAngle                             :FB_BA_Label:=( sObjName:='FDB',sDescr:='Feedback blind angle');
  LblControl_FeedbackSunblindPrio                              :FB_BA_Label:=( sObjName:='FDB',sDescr:='Feedback Telegram-Priority');
// 
  LblControl_TimeDelayStormOn                                  :FB_BA_Label:=( sObjName:='TON',sDescr:='Storm-detection time delay on');
  LblControl_TimeDelayStormOff                                 :FB_BA_Label:=( sObjName:='TOF',sDescr:='Storm-detection time delay off');
  LblControl_MaintenanceEnable                                 :FB_BA_Label:=( sObjName:='EN_',sDescr:='Maintenence positioning enable');
  LblControl_MaintenancePosition                               :FB_BA_Label:=( sObjName:='SP_',sDescr:='Setpoint maintenance position');
  LblControl_MaintenanceAngle                                  :FB_BA_Label:=( sObjName:='SP_',sDescr:='Setpoint maintenance angle');
  LblControl_FacadeThermoAutomaticEnable                       :FB_BA_Label:=( sObjName:='EN_',sDescr:='Facade-Thermoautomatic enable');
  LblControl_FacadeThermoAutomaticCoolingPosition              :FB_BA_Label:=( sObjName:='SP_',sDescr:='Facade-Thermoautomatic cooling-position');
  LblControl_FacadeThermoAutomaticCoolingAngle                 :FB_BA_Label:=( sObjName:='SP_',sDescr:='Facade-Thermoautomatic cooling-angle');
  LblControl_FacadeTwilightAutomaticEnable                     :FB_BA_Label:=( sObjName:='EN_',sDescr:='Facade-Twilightautomatic enable');
  LblControl_SunProtectionValueOn                              :FB_BA_Label:=( sObjName:='SP_',sDescr:='Sun-protection brightness on');
  LblControl_SunProtectionValueOff                             :FB_BA_Label:=( sObjName:='SP_',sDescr:='Sun-protection brightness off');
  LblControl_TimeDelaySunProtectionOn                          :FB_BA_Label:=( sObjName:='TON',sDescr:='Sun-protection brightness on');
  LblControl_TimeDelaySunProtectionOff                         :FB_BA_Label:=( sObjName:='TOF',sDescr:='Sun-protection brightness off');
  LblControl_FacadeParkingEnable                               :FB_BA_Label:=( sObjName:='EN_',sDescr:='Facade-parking enable');
  LblControl_FacadeParkingPosition                             :FB_BA_Label:=( sObjName:='SP_',sDescr:='Facade-parking position');
  LblControl_FacadeParkingAngle                                :FB_BA_Label:=( sObjName:='SP_',sDescr:='Facade-parking angle');
  LblControl_WindProtectionState                               :FB_BA_Label:=( sObjName:='STA',sDescr:='State wind-protection');
  LblControl_SunProtectionState                                :FB_BA_Label:=( sObjName:='STA',sDescr:='State sun-protection');
// 
  LblControl_LowWaterMonitor                                   :FB_BA_Label:=( sObjName:='DST',sDescr:='Low water monitor');
  LblControl_FireAlert                                         :FB_BA_Label:=( sObjName:='DST',sDescr:='Fire alert');
  LblControl_Burglary                                          :FB_BA_Label:=( sObjName:='DST',sDescr:='Burglary alert');
  LblControl_CentralSwitchOff                                  :FB_BA_Label:=( sObjName:='PLS',sDescr:='Central switch-off');
  LblControl_ForcedVentilation                                 :FB_BA_Label:=( sObjName:='PLS',sDescr:='Forced ventilation ');
  LblControl_SmokeExtraction                                   :FB_BA_Label:=( sObjName:='PLS',sDescr:='Smoke extraction');
  LblControl_SetpointIce                                       :FB_BA_Label:=( sObjName:='SP_',sDescr:='Setpoint Ice');
  LblControl_SunProtectionInterval                             :FB_BA_Label:=( sObjName:='SP_',sDescr:='Sun-protection positioning interval');
  LblControl_DeiceTime                                         :FB_BA_Label:=( sObjName:='SP_',sDescr:='Frost-protection deice-time');
  LblControl_GlobalThermoAutomaticValueOn                      :FB_BA_Label:=( sObjName:='SP_',sDescr:='Thermo-automatic radiation-value on');
  LblControl_GlobalThermoAutomaticValueOff                     :FB_BA_Label:=( sObjName:='SP_',sDescr:='Thermo-automatic radiation-value off');
  LblControl_GlobalTwilightAutomaticValueOn                    :FB_BA_Label:=( sObjName:='SP_',sDescr:='Twilight-automatic brightness-value on');
  LblControl_GlobalTwilightAutomaticValueOff                   :FB_BA_Label:=( sObjName:='SP_',sDescr:='Twilight-automatic brightness-value on');
  LblControl_IceAlert                                          :FB_BA_Label:=( sObjName:='DST',sDescr:='Ice alert');
  LblControl_GlobalThermoAutomaticRelease                      :FB_BA_Label:=( sObjName:='EN_',sDescr:='Thermo-automatic release');
  LblControl_GlobalTwilightAutomaticRelease                    :FB_BA_Label:=( sObjName:='EN_',sDescr:='Twilight-automatic release');
  LblControl_GlobalResetManMode                                :FB_BA_Label:=( sObjName:='PLS',sDescr:='Global Reset Manual Mode');
// 
  LblControl_BuildingEnergyLevelManual                         :FB_BA_Label:=( sObjName:='OPS',sDescr:='Building-energy-level manual selection');
  LblControl_BuildingEnergyLevelActual                         :FB_BA_Label:=( sObjName:='POM',sDescr:='Building-energy-level actual selection');
  LblControl_BuildingEnergyLevelSched                          :FB_BA_Label:=( sObjName:='SCH',sDescr:='Building-energy-level scheduler');
  LblControl_BuildingModeManual                                :FB_BA_Label:=( sObjName:='OPS',sDescr:='Building-mode manual selection');
  LblControl_BuildingModeActual                                :FB_BA_Label:=( sObjName:='POM',sDescr:='Building-mode actual selection');
  LblControl_BuildingModeSched                                 :FB_BA_Label:=( sObjName:='SCH',sDescr:='Building-mode scheduler');
// 
  LblControl_SummerCompensationX1                              :FB_BA_Label:=( sObjName:='IPX',sDescr:='Summercompensation X1');
  LblControl_SummerCompensationX2                              :FB_BA_Label:=( sObjName:='IPX',sDescr:='Summercompensation X2');
  LblControl_SummerCompensationY1                              :FB_BA_Label:=( sObjName:='IPY',sDescr:='Summercompensation Y1');
  LblControl_SummerCompensationY2                              :FB_BA_Label:=( sObjName:='IPY',sDescr:='Summercompensation Y2');
  LblControl_WinterCompensationX1                              :FB_BA_Label:=( sObjName:='IPX',sDescr:='Wintercompensation X1');
  LblControl_WinterCompensationX2                              :FB_BA_Label:=( sObjName:='IPX',sDescr:='Wintercompensation X2');
  LblControl_WinterCompensationY1                              :FB_BA_Label:=( sObjName:='IPY',sDescr:='Wintercompensation Y1');
  LblControl_WinterCompensationY2                              :FB_BA_Label:=( sObjName:='IPY',sDescr:='Wintercompensation Y2');
  LblControl_SummerCompensation                                :FB_BA_Label:=( sObjName:='SCP',sDescr:='SummerCompensation');
  LblControl_WinterCompensation                                :FB_BA_Label:=( sObjName:='WCP',sDescr:='WinterCompensation');
  LblControl_SummerCompensationYmin                            :FB_BA_Label:=( sObjName:='SPI',sDescr:='Summer Compensation Ymin');
  LblControl_SummerCompensationYmax                            :FB_BA_Label:=( sObjName:='SPX',sDescr:='Summer Compensation Ymax');
  LblControl_WinterCompensationYmin                            :FB_BA_Label:=( sObjName:='SPI',sDescr:='Winter Compensation Ymin');
  LblControl_WinterCompensationYmax                            :FB_BA_Label:=( sObjName:='SPX',sDescr:='Winter Compensation Ymax');
  LblControl_SummerCompensationSp                              :FB_BA_Label:=( sObjName:='SPC',sDescr:='Summer Compensation Setpoint');
  LblControl_WinterCompensationSp                              :FB_BA_Label:=( sObjName:='SPC',sDescr:='Winter Compensation Setpoint');
  LblControl_SetpointShiftHeating                              :FB_BA_Label:=( sObjName:='SP_',sDescr:='Setpoint shift heating');
  LblControl_SetpointShiftCooling                              :FB_BA_Label:=( sObjName:='SP_',sDescr:='Setpoint shift cooling');
  LblControl_DampConstant                                      :FB_BA_Label:=( sObjName:='SP_',sDescr:='Damp constant');
// 
  LblControl_DelayOn                                           :FB_BA_Label:=( sObjName:='TON',sDescr:='Switch-on delay');
  LblControl_DelayOff                                          :FB_BA_Label:=( sObjName:='TOF',sDescr:='Switch-off delay');
  LblControl_AntiBlocking                                      :FB_BA_Label:=( sObjName:='ABK',sDescr:='Anti Blocking');
  LblControl_IdlePeriod                                        :FB_BA_Label:=( sObjName:='ITV',sDescr:='Idle Period');
  LblControl_ImpulsLength                                      :FB_BA_Label:=( sObjName:='IPL',sDescr:='Impuls length');
  LblControl_SuppyAirTempSetpointHeaterCalc                    :FB_BA_Label:=( sObjName:='SPC',sDescr:='Suppy Air Sp Heater Calc');
  LblControl_SuppyAirTempSetpointCoolerCalc                    :FB_BA_Label:=( sObjName:='SPC',sDescr:='Suppy Air Sp Cooler Calc');
  LblControl_SuppyAirTempSetpointERCCalc                       :FB_BA_Label:=( sObjName:='SPC',sDescr:='Suppy Air Sp ERC Calc');
  LblControl_X01                                               :FB_BA_Label:=( sObjName:='SPX',sDescr:='Value Base [X1]');
  LblControl_X02                                               :FB_BA_Label:=( sObjName:='SPX',sDescr:='Value Base [X2]');
  LblControl_X03                                               :FB_BA_Label:=( sObjName:='SPX',sDescr:='Value Base [X3]');
  LblControl_X04                                               :FB_BA_Label:=( sObjName:='SPX',sDescr:='Value Base [X4]');
  LblControl_X05                                               :FB_BA_Label:=( sObjName:='SPX',sDescr:='Value Base [X5]');
  LblControl_X06                                               :FB_BA_Label:=( sObjName:='SPX',sDescr:='Value Base [X6]');
  LblControl_X07                                               :FB_BA_Label:=( sObjName:='SPX',sDescr:='Value Base [X7]');
  LblControl_Y01                                               :FB_BA_Label:=( sObjName:='SPY',sDescr:='Value Base [Y1]');
  LblControl_Y02                                               :FB_BA_Label:=( sObjName:='SPY',sDescr:='Value Base [Y2]');
  LblControl_Y02_03                                            :FB_BA_Label:=( sObjName:='SPY',sDescr:='Value Base [Y2Y3]');
  LblControl_Y03                                               :FB_BA_Label:=( sObjName:='SPY',sDescr:='Value Base [Y3]');
  LblControl_Y04                                               :FB_BA_Label:=( sObjName:='SPY',sDescr:='Value Base [Y4]');
  LblControl_Y05                                               :FB_BA_Label:=( sObjName:='SPY',sDescr:='Value Base [Y5]');
  LblControl_Y06                                               :FB_BA_Label:=( sObjName:='SPY',sDescr:='Value Base [Y6]');
  LblControl_Y07                                               :FB_BA_Label:=( sObjName:='SPY',sDescr:='Value Base [Y7]');
  LblControl_Feedback                                          :FB_BA_Label:=( sObjName:='FDM',sDescr:='Feedback monitoring');
  LblControl_PreAlarmLimitMAX                                  :FB_BA_Label:=( sObjName:='LMX',sDescr:='Pre Alarm Limit MAX');
  LblControl_PreAlarmLimitMIN                                  :FB_BA_Label:=( sObjName:='LMI',sDescr:='Pre Alarm Limit MIN');
  LblControl_PreAlarmFault                                     :FB_BA_Label:=( sObjName:='DST',sDescr:='Pre Alarm Fault');
  LblControl_MainAlarmLimitMAX                                 :FB_BA_Label:=( sObjName:='LMX',sDescr:='Main Alarm Limit MAX');
  LblControl_MainAlarmLimitMIN                                 :FB_BA_Label:=( sObjName:='LMI',sDescr:='Main Alarm Limit MIN');
  LblControl_MainAlarmFault                                    :FB_BA_Label:=( sObjName:='DST',sDescr:='Main Alarm Fault');
  LblControl_ProcPreRinse                                      :FB_BA_LabelProcess:=( sProcessName:='Process Pre Rinse');
  LblControl_ProjectInfo                                       :FB_BA_Label:=( sObjName:='PI_',sDescr:='Project Info');
END_VAR

// ---- Templates/GVLs/DPAD/Labels/1033/LblFunctions1033.TcGVL
{region '#Template'}
	{attribute 'Version' := '1.0.0.0'}
	{attribute 'Tags' := '"LCID": "1031", "Text": "GVL, AKS, Labels, ObjectName, Description"'}
	{attribute 'Tags' := '"LCID": "1033", "Text": "GVL, DPAD, Labels, ObjectName, Description"'}
	{attribute 'Description' := '"LCID": "1031", "Text": "Anlagenkennzeichnungssystem, Labels functions"'}
	{attribute 'Description' := '"LCID": "1033", "Text": "Data Point Addressing Description, Labels functions"'}
{endregion}

{attribute 'global_init_slot' := '40510'}
VAR_GLOBAL
  LblFunctions_Requirement                                       :FB_BA_Label:=( sObjName:='REQ',sDescr:='Requirement');
  LblFunctions_SystemSwitch                                      :FB_BA_Label:=( sObjName:='PLS',sDescr:='Plant switch');
  LblFunctions_StatusOccupiedRoom                                :FB_BA_Label:=( sObjName:='OCC',sDescr:='Occupied status room');
  LblFunctions_LimitCalculatedValue                              :FB_BA_Label:=( sObjName:='LMC',sDescr:='Calculated limit value');
  LblFunctions_SetpointCalculated                                :FB_BA_Label:=( sObjName:='SPC',sDescr:='Calculated setpoint');
  LblFunctions_ReadyForOperation                                 :FB_BA_Label:=( sObjName:='RFO',sDescr:='Ready for operation');
  LblFunctions_OperationalMessage                                :FB_BA_Label:=( sObjName:='OM_',sDescr:='Operational message');
  LblFunctions_HoursOfOperation                                  :FB_BA_Label:=( sObjName:='OH_',sDescr:='Operating hours');
  LblFunctions_LimitValueHoursOfOperation                        :FB_BA_Label:=( sObjName:='OHL',sDescr:='Operating hours limit value');
  LblFunctions_ObjectCalendar                                    :FB_BA_Label:=( sObjName:='CAL',sDescr:='Calendar object');
  LblFunctions_ObjectCommand                                     :FB_BA_Label:=( sObjName:='COM',sDescr:='Command object');
  LblFunctions_DifferentialConstantController                    :FB_BA_Label:=( sObjName:='TV_',sDescr:='Differential constant controller');
  LblFunctions_SwitchOnErrorUnauthorisedON                       :FB_BA_Label:=( sObjName:='SWE',sDescr:='Switch-on error, unauthorised ON');
  LblFunctions_EnergyLevel                                       :FB_BA_Label:=( sObjName:='EL_',sDescr:='Energy level');
  LblFunctions_EnergyLevelCalculated                             :FB_BA_Label:=( sObjName:='ELC',sDescr:='Energy level calculated');
  LblFunctions_UnlockingDevice                                   :FB_BA_Label:=( sObjName:='UNL',sDescr:='Unlocking device');
  LblFunctions_ObjectEventEnrollment                             :FB_BA_Label:=( sObjName:='EE_',sDescr:='Event enrollment object');
  LblFunctions_Enabled                                           :FB_BA_Label:=( sObjName:='EN_',sDescr:='Enabled');
  LblFunctions_DangerAlarm                                       :FB_BA_Label:=( sObjName:='DA_',sDescr:='Danger alarm');
  LblFunctions_Threshold                                         :FB_BA_Label:=( sObjName:='LM_',sDescr:='Limit value');
  LblFunctions_LimitMAX                                          :FB_BA_Label:=( sObjName:='LMX',sDescr:='MAX limit');
  LblFunctions_LimitMIN                                          :FB_BA_Label:=( sObjName:='LMI',sDescr:='MIN limit');
  LblFunctions_LimitNight                                        :FB_BA_Label:=( sObjName:='LMN',sDescr:='Night limit');
  LblFunctions_LimitDay                                          :FB_BA_Label:=( sObjName:='LMD',sDescr:='Day limit');
  LblFunctions_ObjectGroup                                       :FB_BA_Label:=( sObjName:='GP_',sDescr:='Group object');
  LblFunctions_localPriorityAndOperatingUnitsManualMessage       :FB_BA_Label:=( sObjName:='MNM',sDescr:='local priority and operating units manual message');
  LblFunctions_HeatingCharacteristicCurveExponent                :FB_BA_Label:=( sObjName:='HEX',sDescr:='Heating characteristic curve exponent');
  LblFunctions_HeatingCharacteristicCurveParallelDisplacement    :FB_BA_Label:=( sObjName:='HPD',sDescr:='Heating characteristic curve parallel displacement');
  LblFunctions_HeatingCharacteristicCurveSteepness               :FB_BA_Label:=( sObjName:='HST',sDescr:='Heating characteristic curve steepness');
  LblFunctions_HeatingCircuitNightReduction                      :FB_BA_Label:=( sObjName:='NGT',sDescr:='Heating circuit night reduction');
  LblFunctions_Hysteresis                                        :FB_BA_Label:=( sObjName:='HYS',sDescr:='Hysteresis');
  LblFunctions_Calendar                                          :FB_BA_Label:=( sObjName:='CAL',sDescr:='Calendar');
  LblFunctions_RuntimeError                                      :FB_BA_Label:=( sObjName:='RUN',sDescr:='Runtime error');
  LblFunctions_LoopMAXLimit                                      :FB_BA_Label:=( sObjName:='LPX',sDescr:='Loop MAX limit');
  LblFunctions_LoopMINLimit                                      :FB_BA_Label:=( sObjName:='LPI',sDescr:='Loop MIN limit');
  LblFunctions_LoopObject                                        :FB_BA_Label:=( sObjName:='LP_',sDescr:='Loop object (controller object) – complex object');
  LblFunctions_LoopObjectCascadeSupplyAirTemperature             :FB_BA_Label:=( sObjName:='LP_',sDescr:='Cascade controller supply air temperature ');
  LblFunctions_LoopObjectCascadeSupplyAirHumidity                :FB_BA_Label:=( sObjName:='LP_',sDescr:='Cascade controller supply air humidity ');
  LblFunctions_MaximumValue                                      :FB_BA_Label:=( sObjName:='MAX',sDescr:='Maximum value');
  LblFunctions_MeasuredValue                                     :FB_BA_Label:=( sObjName:='MV_',sDescr:='Measured value');
  LblFunctions_MeasuredValueCalculated                           :FB_BA_Label:=( sObjName:='MVC',sDescr:='Measured value calculated');
  LblFunctions_MeasuredValueEast                                 :FB_BA_Label:=( sObjName:='MV_',sDescr:='Measured value East');
  LblFunctions_MeasuredValueNorth                                :FB_BA_Label:=( sObjName:='MV_',sDescr:='Measured value North');
  LblFunctions_MeasuredValueSouth                                :FB_BA_Label:=( sObjName:='MV_',sDescr:='Measured value South');
  LblFunctions_MeasuredValueWest                                 :FB_BA_Label:=( sObjName:='MV_',sDescr:='Measured value West');
  LblFunctions_MinimumValue                                      :FB_BA_Label:=( sObjName:='MIN',sDescr:='Minimum value');
  LblFunctions_Mean                                              :FB_BA_Label:=( sObjName:='MVL',sDescr:='Mean value');
  LblFunctions_FollowUpTime                                      :FB_BA_Label:=( sObjName:='FUT',sDescr:='Follow-up time');
  LblFunctions_ResetTime                                         :FB_BA_Label:=( sObjName:='RST',sDescr:='Reset time');
  LblFunctions_FeedbackDelay                                     :FB_BA_Label:=( sObjName:='TDF',sDescr:='Time delay feedback');
  LblFunctions_ObjectNotificationClass                           :FB_BA_Label:=( sObjName:='NC_',sDescr:='Notification class object');
  LblFunctions_EventClassObject                                  :FB_BA_Label:=( sObjName:='ECL',sDescr:='Event class');
  LblFunctions_Programobject                                     :FB_BA_Label:=( sObjName:='PRG',sDescr:='Program');
  LblFunctions_ProportionalBand                                  :FB_BA_Label:=( sObjName:='XP_',sDescr:='Proportional band');
  LblFunctions_FeedbackOPEN                                      :FB_BA_Label:=( sObjName:='FDO',sDescr:='Feedback OPEN');
  LblFunctions_FeedbackCLOSED                                    :FB_BA_Label:=( sObjName:='FDC',sDescr:='Feedback CLOSED');
  LblFunctions_FeedbackValue                                     :FB_BA_Label:=( sObjName:='FDB',sDescr:='Feedback value');
  LblFunctions_FeedbackErrorOPEN                                 :FB_BA_Label:=( sObjName:='FEO',sDescr:='Feedback error OPEN');
  LblFunctions_FeedbackErrorCLOSED                               :FB_BA_Label:=( sObjName:='FEC',sDescr:='Feedback error CLOSED');
  LblFunctions_Feedback                                          :FB_BA_Label:=( sObjName:='FDB',sDescr:='Feedback');
  LblFunctions_ExecutionControl                                  :FB_BA_Label:=( sObjName:='EXC',sDescr:='Execution control');
  LblFunctions_SwitchingCommand                                  :FB_BA_Label:=( sObjName:='SC_',sDescr:='Switching command');
  LblFunctions_Scheduler                                         :FB_BA_Label:=( sObjName:='SCH',sDescr:='Scheduler');
  LblFunctions_Setpoint                                          :FB_BA_Label:=( sObjName:='SP_',sDescr:='Setpoint');
  LblFunctions_SetpointComfortHeating                            :FB_BA_Label:=( sObjName:='SP_',sDescr:='Setpoint comfort heating');
  LblFunctions_SetpointPreComfortHeating                         :FB_BA_Label:=( sObjName:='SP_',sDescr:='Setpoint pre-comfort heating');
  LblFunctions_SetpointEconomyHeating                            :FB_BA_Label:=( sObjName:='SP_',sDescr:='Setpoint economy heating');
  LblFunctions_SetpointProtectionHeating                         :FB_BA_Label:=( sObjName:='SP_',sDescr:='Setpoint protection heating');
  LblFunctions_SetpointComfortCooling                            :FB_BA_Label:=( sObjName:='SP_',sDescr:='Setpoint comfort cooling');
  LblFunctions_SetpointPreComfortCooling                         :FB_BA_Label:=( sObjName:='SP_',sDescr:='Setpoint pre-comfort cooling');
  LblFunctions_SetpointEconomyCooling                            :FB_BA_Label:=( sObjName:='SP_',sDescr:='Setpoint economy cooling');
  LblFunctions_SetpointProtectionCooling                         :FB_BA_Label:=( sObjName:='SP_',sDescr:='Setpoint protection cooling');
  LblFunctions_SetpointBase                                      :FB_BA_Label:=( sObjName:='SPB',sDescr:='Base setpoint');
  LblFunctions_SetpointHeating                                   :FB_BA_Label:=( sObjName:='SPH',sDescr:='Heating setpoint');
  LblFunctions_SetpointCooling                                   :FB_BA_Label:=( sObjName:='SPC',sDescr:='Cooling setpoint');
  LblFunctions_SetpointMaximum                                   :FB_BA_Label:=( sObjName:='SPX',sDescr:='Setpoint, maximum');
  LblFunctions_SetpointMechanical                                :FB_BA_Label:=( sObjName:='SPM',sDescr:='Setpoint, mechanical');
  LblFunctions_SetpointMinimum                                   :FB_BA_Label:=( sObjName:='SPI',sDescr:='Setpoint, minimum');
  LblFunctions_SetpointNight                                     :FB_BA_Label:=( sObjName:='SPN',sDescr:='Night setpoint');
  LblFunctions_SetpointDay                                       :FB_BA_Label:=( sObjName:='SPD',sDescr:='Day setpoint');
  LblFunctions_SetpointAdjuster                                  :FB_BA_Label:=( sObjName:='SPA',sDescr:='Setpoint adjuster');
  LblFunctions_SetpointAdjustmentMechanical                      :FB_BA_Label:=( sObjName:='SPA',sDescr:='Setpoint adjustment, mechanical');
  LblFunctions_Selection                                         :FB_BA_Label:=( sObjName:='SEL',sDescr:='Selection');
  LblFunctions_Status                                            :FB_BA_Label:=( sObjName:='STA',sDescr:='Status');
  LblFunctions_ControlSignal                                     :FB_BA_Label:=( sObjName:='CS_',sDescr:='Control signal');
  LblFunctions_Fault                                             :FB_BA_Label:=( sObjName:='FAU',sDescr:='Fault');
  LblFunctions_FaultFuse                                         :FB_BA_Label:=( sObjName:='FAU',sDescr:='Fuse fault ');
  LblFunctions_Button                                            :FB_BA_Label:=( sObjName:='BUT',sDescr:='Button');
  LblFunctions_DeadZone                                          :FB_BA_Label:=( sObjName:='DZ_',sDescr:='Dead zone');
  LblFunctions_ObjectTrendLogMultiple                            :FB_BA_Label:=( sObjName:='TRM',sDescr:='Trend log multiple object');
  LblFunctions_ObjectTrendLog                                    :FB_BA_Label:=( sObjName:='TR_',sDescr:='Trend log object');
  LblFunctions_AmplificationController                           :FB_BA_Label:=( sObjName:='KP_',sDescr:='Amplification controller');
  LblFunctions_RetentionPeriod                                   :FB_BA_Label:=( sObjName:='TV_',sDescr:='Retention period');
  LblFunctions_MaintenanceMessage                                :FB_BA_Label:=( sObjName:='MTM',sDescr:='Maintenance message');
  LblFunctions_Efficiency                                        :FB_BA_Label:=( sObjName:='EFC',sDescr:='Efficiency');
  LblFunctions_CountValue                                        :FB_BA_Label:=( sObjName:='CNT',sDescr:='Count value');
  LblFunctions_TimeProgram                                       :FB_BA_Label:=( sObjName:='TPR',sDescr:='Time program');
// Beckhoff Scale
  LblFunctions_ValueX1                                           :FB_BA_Label:=( sObjName:='IPX',sDescr:='Value interpolation point [X1]');
  LblFunctions_ValueX2                                           :FB_BA_Label:=( sObjName:='IPX',sDescr:='Value interpolation point [X2]');
  LblFunctions_ValueX3                                           :FB_BA_Label:=( sObjName:='IPX',sDescr:='Value interpolation point [X3]');
  LblFunctions_ValueX4                                           :FB_BA_Label:=( sObjName:='IPX',sDescr:='Value interpolation point [X4]');
  LblFunctions_ValueX5                                           :FB_BA_Label:=( sObjName:='IPX',sDescr:='Value interpolation point [X4]');
  LblFunctions_ValueX6                                           :FB_BA_Label:=( sObjName:='IPX',sDescr:='Value interpolation point [X4]');
  LblFunctions_ValueX7                                           :FB_BA_Label:=( sObjName:='IPX',sDescr:='Value interpolation point [X4]');
  LblFunctions_ValueY1                                           :FB_BA_Label:=( sObjName:='IPY',sDescr:='Value interpolation point [Y1]');
  LblFunctions_ValueY2                                           :FB_BA_Label:=( sObjName:='IPY',sDescr:='Value interpolation point [Y2]');
  LblFunctions_ValueY3                                           :FB_BA_Label:=( sObjName:='IPY',sDescr:='Value interpolation point [Y3]');
  LblFunctions_ValueY2_3                                         :FB_BA_Label:=( sObjName:='IPY',sDescr:='Value interpolation point [Y2-Y3]');
  LblFunctions_ValueY4                                           :FB_BA_Label:=( sObjName:='IPY',sDescr:='Value interpolation point [Y4]');
  LblFunctions_ValueY5                                           :FB_BA_Label:=( sObjName:='IPY',sDescr:='Value interpolation point [Y4]');
  LblFunctions_ValueY6                                           :FB_BA_Label:=( sObjName:='IPY',sDescr:='Value interpolation point [Y4]');
  LblFunctions_ValueY7                                           :FB_BA_Label:=( sObjName:='IPY',sDescr:='Value interpolation point [Y4]');
  LblFunctions_SuppyAirTempSetpointHeaterCalc                    :FB_BA_Label:=( sObjName:='SPC',sDescr:='Supply air Temperature setpoint heater calculated');
  LblFunctions_SuppyAirTempSetpointCoolerCalc                    :FB_BA_Label:=( sObjName:='SPC',sDescr:='Supply air Temperature setpoint cooler calculated');
  LblFunctions_SuppyAirTempSetpointERCCalc                       :FB_BA_Label:=( sObjName:='SPC',sDescr:='Supply air Temperature setpoint ERC calculated');
END_VAR

// ---- Templates/GVLs/DPAD/Labels/Composition/LblCmpAC.TcGVL
{region '#Template'}
	{attribute 'Version' := '1.0.0.0'}
	{attribute 'Tags' := '"LCID": "1031", "Text": "GVL, AC, AKS, Plants, ObjectName, Description"'}
	{attribute 'Tags' := '"LCID": "1033", "Text": "GVL, AC, DPAD, Plants, ObjectName, Description"'}
	{attribute 'Description' := '"LCID": "1031", "Text": "Anlagenkennzeichnungssystem, AC Labels Kompensation"'}
	{attribute 'Description' := '"LCID": "1033", "Text": "Data Point Addressing Description, AC labels compensation"'}
{endregion}

{attribute 'qualified_only'}
VAR_GLOBAL
///////////////////////
//	Aggregates\Cooler	
	Cooler_TFl							:FB_BA_Label	:= LblAggregates_TemperatureFlow;	
	Cooler_TRt							:FB_BA_Label	:= LblAggregates_TemperatureReturnFlow;	

	Cooler_TSuACtrl						:FB_BA_Label	:= LblControl_SupplyAirTemperatureControl;
	Cooler_TSuACtrl_Ctrl				:FB_BA_Label	:= LblFunctions_LoopObject; 
	Cooler_TSuALimitationCtrl			:FB_BA_Label	:= LblControl_SupplyAirTemperatureLimitationControl;

	Cooler_XSuACtrl						:FB_BA_Label	:= LblControl_SupplyAirDehumidifierControl; 
	Cooler_XSuACtrl_Ctrl				:FB_BA_Label	:= LblFunctions_LoopObject; 
	Cooler_Dehumf						:FB_BA_Label	:= LblControl_OperationalMessageDehumidification;	

	Cooler_Vlv							:FB_BA_Label	:= LblAggregates_Valve;
	Cooler_Pu							:FB_BA_Label	:= LblAggregates_Pump;
	
//	Aggregates\ERC
	ERC_DiffPrssSwi						:FB_BA_Label	:= LblAggregates_PressureDifferential;												 										 
	ERC_IcePrtcRamp						:FB_BA_Label	:= LblControl_EnergyRecoveryDeicingRamp;
	ERC_Motor							:FB_BA_Label	:= LblAggregates_HeatRecovery;
	ERC_TExhACtrl						:FB_BA_Label	:= LblControl_ExhaustAirTemperatureControl;
	ERC_TSuACtrl						:FB_BA_Label	:= LblControl_SupplyAirTemperatureControl;
	ERC_TSuACtrl_Ctrl					:FB_BA_Label	:= LblFunctions_LoopObject; 

	ERC_DiffPrssSensor					:FB_BA_Label	:= LblAggregates_PressureDifferential;	
	ERC_Damping							:FB_BA_Label	:= LblAggregates_PressureDifferential;
	ERC_IcePrtcDiffPrssCtrl				:FB_BA_Label	:= LblControl_ExhaustAirTemperatureControl;
	ERC_Dmp								:FB_BA_Label	:= LblAggregates_VentilationDamperSupplyAir;	
	ERC_ByDmp							:FB_BA_Label	:= LblAggregates_VentilationDamperBypassAir;

//	Aggregates\Humidifier
	Humf_HuDet							:FB_BA_Label	:= LblAggregates_Hygrostat;	
//////////////////////
	Humf_Dst							:FB_BA_Label	:= LblAggregates_Airwasher;			
	Humf_Dst_Input						:FB_BA_Label	:= LblFunctions_Fault;			
	Humf_LowWaterMonitor				:FB_BA_Label	:= LblAggregates_Airwasher;			
	Humf_LowWaterMonitor_Input			:FB_BA_Label	:= LblControl_LowWaterMonitor;	
	Humf_ReadyOp						:FB_BA_Label	:= LblAggregates_Airwasher;			
	Humf_ReadyOp_Input					:FB_BA_Label	:= LblFunctions_ReadyForOperation;			
	Humf_MntnSwi						:FB_BA_Label	:= LblAggregates_Airwasher;			
	Humf_MntnSwi_Input					:FB_BA_Label	:= LblFunctions_MaintenanceMessage;
//////////////////////	
	Humf_AirWasher						:FB_BA_Label	:= LblAggregates_Airwasher;			
	Humf_AirWasher_Dst					:FB_BA_Label	:= LblFunctions_Fault;			
	Humf_AirWasher_LowWaterMonitor		:FB_BA_Label	:= LblControl_LowWaterMonitor;	
	Humf_AirWasher_ReadyOp				:FB_BA_Label	:= LblFunctions_ReadyForOperation;			
	Humf_AirWasher_MntnSwi				:FB_BA_Label	:= LblFunctions_MaintenanceMessage;				
	
	Humf_XSuACtrl						:FB_BA_Label	:= LblControl_SupplyAirHumidifierController;
	Humf_XSuACtrl_Ctrl					:FB_BA_Label	:= LblFunctions_LoopObject; 
	Humf_Vlv							:FB_BA_Label	:= LblAggregates_Valve;
	Humf_Pu								:FB_BA_Label	:= LblAggregates_Pump;			
	Humf_DlyOff							:FB_BA_Label	:= LblControl_DelayOff;	

	Humf_HLmtCtrl						:FB_BA_Label	:= LblControl_HumidityLimitationControl;

//	Aggregates\MixedAir
	Mix_TSuACtrl						:FB_BA_Label	:= LblControl_SupplyAirTemperatureControl;
	Mix_TSuACtrl_Ctrl					:FB_BA_Label	:= LblFunctions_LoopObject; 
	Mix_StartUpRamp						:FB_BA_Label	:= LblControl_MixedAirStartUpRamp;
	Mix_DmpMixA							:FB_BA_Label	:= LblAggregates_VentilationDamperMixAir;	
	Mix_DmpOuA							:FB_BA_Label	:= LblAggregates_VentilationDamperOutsideAir;	
	Mix_DmpExhA							:FB_BA_Label	:= LblAggregates_VentilationDamperExhaustAir;	

//	Aggregates\pre-heater
	PreHtr_TFl							:FB_BA_Label	:= LblAggregates_TemperatureFlow;	
	PreHtr_TRt							:FB_BA_Label	:= LblAggregates_TemperatureReturnFlow;	
	PreHtr_TSuACtrl						:FB_BA_Label	:= LblControl_SupplyAirTemperatureControl;
	PreHtr_TSuACtrl_Ctrl				:FB_BA_Label	:= LblFunctions_LoopObject; 
	PreHtr_TFrost						:FB_BA_Label	:= LblControl_TemperatureFrost;	
	PreHtr_TFrostPrtcCtrlAir			:FB_BA_Label	:= LblControl_FrostProtectionControl;
	PreHtr_FrostThermostat				:FB_BA_Label	:= LblAggregates_FrostProtectionMonitor;												 										 
	PreHtr_FrostThermostat_Input		:FB_BA_Label	:= LblFunctions_DangerAlarm;
	PreHtr_Vlv							:FB_BA_Label	:= LblAggregates_Valve;
	PreHtr_Pu							:FB_BA_Label	:= LblAggregates_Pump;		
	PreHtr_TRtCtrl						:FB_BA_Label	:= LblControl_ReturnWaterControl;
	PreHtr_TRtCtrl_SpTRtW				:FB_BA_Label	:= LblFunctions_Setpoint;
	PreHtr_TRtCtrl_PreRinseDelay		:FB_BA_Label	:= LblControl_DelayOn;
	PreHtr_TRtCtrl_PreRinseDelay_TiDly	:FB_BA_Label	:= LblControl_PreRinseDuration;
	PreHtr_TRtCtrl_PreRinseDst			:FB_BA_Label	:= LblControl_DisturbancePreRinse;	 								 
	PreHtr_TRtCtrl_PreRinseSp			:FB_BA_Label	:= LblControl_CalculationPreRinseSetpoint;			
	PreHtr_TRtCtrl_Ctrl					:FB_BA_Label	:= LblFunctions_LoopObject; 		
	
	PreHtr_ProcessPreRinse				:FB_BA_LabelProcess	:= LblControl_ProcPreRinse;

//	Aggregates\re-heater
	ReHtr_TFl							:FB_BA_Label	:= LblAggregates_TemperatureFlow;	
	ReHtr_TRt							:FB_BA_Label	:= LblAggregates_TemperatureReturnFlow;	
	ReHtr_TSuACtrl						:FB_BA_Label	:= LblControl_SupplyAirTemperatureControl;
	ReHtr_TSuACtrl_Ctrl					:FB_BA_Label	:= LblFunctions_LoopObject;
	ReHtr_TMinSuACtrl					:FB_BA_Label	:= LblControl_SupplyAirTemperatureLimitationControl;
 
	ReHtr_Vlv							:FB_BA_Label	:= LblAggregates_Valve;
	ReHtr_Pu							:FB_BA_Label	:= LblAggregates_Pump;		
		
///////////////////////
//	General
	General_OpModMan					:FB_BA_Label	:= LblControl_OperationModeSelection;							
	General_Sched						:FB_BA_Label	:= LblFunctions_Scheduler;							
	General_OpModPr						:FB_BA_Label	:= LblControl_PresentOperationMode;		
	
//	Summer night cooling
	General_SumNgtCol_WthTLoLmt			:FB_BA_Label	:= LblControl_OutsideTemperatureLowLimit;			
	General_SumNgtCol_RmTHys			:FB_BA_Label	:= LblControl_HysteresisRoomTemperature;			
	General_SumNgtCol_SwiOnDiffT		:FB_BA_Label	:= LblControl_OnValueDifferenceOutsideInsightTemperature;			
	General_SumNgtCol_SwiOffDiffT		:FB_BA_Label	:= LblControl_OffValueDifferenceOutsideInsightTemperature;			
	General_SumNgtCol_Q					:FB_BA_Label	:= LblFunctions_OperationalMessage;												 
	General_SumNgtCol_Sched				:FB_BA_Label	:= LblFunctions_Scheduler;		
///////////////////////
//	Setpoint\Temperature
	SpTRm_X1							:FB_BA_Label	:= LblControl_X01;	
	SpTRm_X2							:FB_BA_Label	:= LblControl_X02;	
	SpTRm_X3							:FB_BA_Label	:= LblControl_X03;	
	SpTRm_X4							:FB_BA_Label	:= LblControl_X04;	
	
	SpTRm_Y1							:FB_BA_Label	:= LblControl_Y01;
	SpTRm_Y2_3							:FB_BA_Label	:= LblControl_Y02_03;
	SpTRm_Y4							:FB_BA_Label	:= LblControl_Y03;
	SpTRm_Sp							:FB_BA_Label	:= LblFunctions_SetpointCalculated;
	
	SpTRm_SpColX1						:FB_BA_Label	:= LblControl_SummerCompensationX1;	
	SpTRm_SpColX2						:FB_BA_Label	:= LblControl_SummerCompensationX2;	
	SpTRm_SpColY1						:FB_BA_Label	:= LblControl_SummerCompensationY1;	
	SpTRm_SpColY2						:FB_BA_Label	:= LblControl_SummerCompensationY2;	
	SpTRm_SpColYMin						:FB_BA_Label	:= LblControl_SummerCompensationYmin;
	SpTRm_SpColYMax						:FB_BA_Label	:= LblControl_SummerCompensationYmax;	
	SpTRm_SpCol							:FB_BA_Label	:= LblControl_SummerCompensationSp;	
	
	SpTRm_SpHtgX1						:FB_BA_Label	:= LblControl_WinterCompensationX1;	
	SpTRm_SpHtgX2						:FB_BA_Label	:= LblControl_WinterCompensationX2;	
	SpTRm_SpHtgY1						:FB_BA_Label	:= LblControl_WinterCompensationY1;	
	SpTRm_SpHtgY2						:FB_BA_Label	:= LblControl_WinterCompensationY2;	
	SpTRm_SpHtgYMin						:FB_BA_Label	:= LblControl_WinterCompensationYmin;
	SpTRm_SpHtgYMax						:FB_BA_Label	:= LblControl_WinterCompensationYmax;		
	SpTRm_SpHtg							:FB_BA_Label	:= LblControl_WinterCompensationSp;	
	
	SpTSuA_SelSpErc						:FB_BA_Label	:= LblControl_OperationModeSelection;							
	SpTSuA_SpErc						:FB_BA_Label	:= LblFunctions_SetpointCalculated;	

	TCasCtrl_SpHtg						:FB_BA_Label	:= LblControl_SuppyAirTempSetpointHeaterCalc;			
	TCasCtrl_SpCol						:FB_BA_Label	:= LblControl_SuppyAirTempSetpointCoolerCalc;			
	TCasCtrl_SpErc						:FB_BA_Label	:= LblControl_SuppyAirTempSetpointERCCalc;			
	TCasCtrl_Ctrl						:FB_BA_Label	:= LblFunctions_LoopObjectCascadeSupplyAirTemperature; 			
	TCasCtrl_SelSpErc					:FB_BA_Label	:= LblControl_OperationModeSelection;							
//	Setpoint\Humidity
	HumCasCtrl_Ctrl						:FB_BA_Label	:= LblFunctions_LoopObjectCascadeSupplyAirHumidity; 	
	SpHum_SpH							:FB_BA_Label	:= LblControl_SetpointRelHumidity;			
	SpHum_SpX							:FB_BA_Label	:= LblControl_SetpointAbsHumidity;
	SpHum_SpHHumf						:FB_BA_Label	:= LblControl_SetpointRelHumidityHumidification;			
	SpHum_SpHDehumf						:FB_BA_Label	:= LblControl_SetpointRelHumidityDehumidification;			
	SpHum_SpXHumf						:FB_BA_Label	:= LblControl_SetpointAbsHumidityHumidification;	
	SpHum_SpXDehumf						:FB_BA_Label	:= LblControl_SetpointAbsHumidityDehumidification;
//	
	PlantControlStatus   	:FB_BA_Label2x :=(iAggregate:=LblControl_PlantControl,		iFunction:=LblFunctions_Status);
	TSequenceControlStatus  :FB_BA_Label2x :=(iAggregate:=LblControl_TSequenceControl,	iFunction:=LblFunctions_Status);		
	HSequenceControlStatus  :FB_BA_Label2x :=(iAggregate:=LblControl_HSequenceControl,	iFunction:=LblFunctions_Status);		
//	AHU	
	AHU_TOuA						:FB_BA_Label	:= LblAggregates_TemperatureOutside;
	AHU_HOuA						:FB_BA_Label	:= LblAggregates_RelativeHumidityOutsideAir;
	AHU_XOuA						:FB_BA_Label	:= LblAggregates_AbsoluteHumidtiyOutsideAir;
	AHU_TExhA						:FB_BA_Label	:= LblAggregates_TemperatureExhaustAir;	
	AHU_HExhA						:FB_BA_Label	:= LblAggregates_RelativeHumidityExhaustAir;	
	AHU_XExhA						:FB_BA_Label	:= LblAggregates_AbsoluteHumidtiyExhaustAir;	
	AHU_TSuA						:FB_BA_Label	:= LblAggregates_TemperatureSupplyAir;	
	AHU_HSuA						:FB_BA_Label	:= LblAggregates_RelativeHumiditySupplyAir;	
	AHU_XSuA						:FB_BA_Label	:= LblAggregates_AbsoluteHumiditySupplyAir;	
	AHU_TExtA						:FB_BA_Label	:= LblAggregates_TemperatureExtractAir;	
	AHU_HExtA						:FB_BA_Label	:= LblAggregates_RelativeHumiditiyExtractAir;	
	AHU_XExtA						:FB_BA_Label	:= LblAggregates_AbsoluteHumidityExtractAir;	
	AHU_TRm							:FB_BA_Label	:= LblAggregates_TemperatureRoomAir;	
	AHU_HRm							:FB_BA_Label	:= LblAggregates_RelativeHumidityRoomHumidity;	
	AHU_XRm							:FB_BA_Label	:= LblAggregates_AbsoluteHumidityRoomAir;	
	AHU_DiffPrssOuAFilt				:FB_BA_Label	:= LblAggregates_PressureDifferentialOutsideAirFilter;	
	AHU_FiltOuAMonit				:FB_BA_Label	:= LblAggregates_AirFilterOutsideAir;
	AHU_DiffPrssExtAFilt			:FB_BA_Label	:= LblAggregates_PressureDifferentialExtractAirFilter;	
	AHU_FiltExtAMonit				:FB_BA_Label	:= LblAggregates_AirFilterExtractAir;
	AHU_SumNgtCol					:FB_BA_Label	:= LblControl_SummerNightCooling;
	AHU_OpMod						:FB_BA_Label	:= LblControl_OperationMode;
	AHU_OuADmp						:FB_BA_Label	:= LblAggregates_VentilationDamperOutsideAir;
	AHU_SuAPrss						:FB_BA_Label	:= LblAggregates_PressureSupplyAir;	
	AHU_SuADiffPrss					:FB_BA_Label	:= LblAggregates_PressureDifferentialSupplyAirFan;	
	AHU_SuAFan						:FB_BA_Label	:= LblAggregates_FanSupplyAir;
	AHU_SuADiffPrssMonit			:FB_BA_Label	:= LblControl_DifferencePressureMonitoringSupplyAirFan;
	AHU_ExhADmp						:FB_BA_Label	:= LblAggregates_VentilationDamperExhaustAir;
	AHU_ExtAPrss					:FB_BA_Label	:= LblAggregates_PressureExtractAir;	
	AHU_ExtADiffPrss				:FB_BA_Label	:= LblAggregates_PressureDifferentialExtractAirFan;	
	AHU_ExtAFan						:FB_BA_Label	:= LblAggregates_FanExtractAir;
	AHU_ExtADiffPrssMonit			:FB_BA_Label	:= LblControl_DifferencePressureMonitoringExtractAirFan;
	AHU_SpTRm						:FB_BA_Label	:= LblControl_TSetpointCalculation;
	AHU_TCasCtrl					:FB_BA_Label	:= LblControl_TCascadeSupplyAirControl;
	AHU_TSeqLink					:FB_BA_Label2x	:= TSequenceControlStatus;
	AHU_SpHRm						:FB_BA_Label	:= LblControl_HSetpointCalculation;
	AHU_HCasCtrl					:FB_BA_Label	:= LblControl_HCascadeSupplyAirControl;
	AHU_HSeqLink					:FB_BA_Label2x	:= HSequenceControlStatus;	
	AHU_ReHtr						:FB_BA_Label	:= LblControl_ReHeater;
	AHU_PreHtr						:FB_BA_Label	:= LblControl_PreHeater;
	AHU_Erc							:FB_BA_Label	:= LblControl_EnergyRecovery;
	AHU_Col							:FB_BA_Label	:= LblControl_Cooler;
	AHU_Humf						:FB_BA_Label	:= LblAggregates_Humidifier;
	AHU_PlantCtrl					:FB_BA_Label2x	:= PlantControlStatus;	



	
END_VAR

// ---- Templates/GVLs/DPAD/Labels/Composition/LblCmpGeneral.TcGVL
{region '#Template'}
	{attribute 'Version' := '1.0.0.0'}
	{attribute 'Tags' := '"LCID": "1031", "Text": "GVL, General, AKS, Plants, ObjectName, Description"'}
	{attribute 'Tags' := '"LCID": "1033", "Text": "GVL, General, DPAD, Plants, ObjectName, Description"'}
	{attribute 'Description' := '"LCID": "1031", "Text": "Anlagenkennzeichnungssystem, Allgemein Labels Kompensation"'}
	{attribute 'Description' := '"LCID": "1033", "Text": "Data Point Addressing Description, General labels compensation"'}
{endregion}

{attribute 'qualified_only'}
VAR_GLOBAL
	BuildingAlarms_FireAlert						: FB_BA_Label := LblControl_FireAlert;
	BuildingAlarms_Bgly								: FB_BA_Label := LblControl_Burglary;
	BuildingAlarms_CentSwiOff						: FB_BA_Label := LblControl_CentralSwitchOff;
                                  				
	BuildingMode_OpModMan							: FB_BA_Label := LblControl_BuildingModeManual;
	BuildingMode_OpModPr							: FB_BA_Label := LblControl_BuildingModeActual;
	BuildingMode_Sched								: FB_BA_Label := LblControl_BuildingModeSched;
                                  				
	BuildingGlobal_BuildAlm							: FB_BA_Label := LblControl_BuildingAlarms;
	BuildingGlobal_BuildMode						: FB_BA_Label := LblControl_BuildingMode;
	
	ControlCabinet_Fuse								: FB_BA_Label := LblControl_Fuse;	
	ControlCabinet_Fuse_Input						: FB_BA_Label := LblFunctions_Fault;	
	ControlCabinet_LampFault						: FB_BA_Label := LblControl_EventIndicationLamp;			
	ControlCabinet_LampFault_Cmd					: FB_BA_Label := LblFunctions_SwitchingCommand;			
	ControlCabinet_AckButton 						: FB_BA_Label := LblControl_Acknowledge;	
	ControlCabinet_AckButton_Input					: FB_BA_Label := LblControl_ButtonLocalAcknowledgement;
	ControlCabinet_AckButton_Value					: FB_BA_Label := LblControl_ButtonRemoteAcknowledgement;
	ControlCabinet_RstHw							: FB_BA_Label := LblControl_AcknowledgeCommand;			
	ControlCabinet_RstHw_Cmd						: FB_BA_Label := LblFunctions_SwitchingCommand;	
	
	EvtGroups_LifeSafety							: FB_BA_Label := LblControl_EvtCategoryLifeSafty;									  
	EvtGroups_AlarmTechnical						: FB_BA_Label := LblControl_EvtCategoryAlarmTechnical;									  
	EvtGroups_Disturbance							: FB_BA_Label := LblControl_EvtCategoryDisturbance;									  
	EvtGroups_Maintenance							: FB_BA_Label := LblControl_EvtCategoryMaintenance;									  
	EvtGroups_Notification							: FB_BA_Label := LblControl_EvtCategoryNotification;									  
	EvtGroups_Other									: FB_BA_Label := LblControl_EvtCategoryOther;									  
	
	Settings_WthParam								: FB_BA_Label := LblControl_WeatherParameters;	
	
	WthParam_SpFrstProtec							: FB_BA_Label := LblControl_SetpointFrostProtection;
	WthParam_TWthLowLimitVal						: FB_BA_Label := LblControl_SetpointMinimumOutsideTemperature;
	WthParam_TWthLowLimit							: FB_BA_Label := LblControl_OperationalMessageTemperatureWeatherLowLimit;	
	WthParam_TWthDamped								: FB_BA_Label := LblControl_MeanDamped;
	WthParam_TWthDampedLowLimit						: FB_BA_Label := LblControl_OperationalMessageTemperatureWeatherDampedLowLimit;	
END_VAR

// ---- Templates/GVLs/DPAD/Labels/Composition/LblCmpHeating.TcGVL
{region '#Template'}
	{attribute 'Version' := '1.0.0.0'}
	{attribute 'Tags' := '"LCID": "1031", "Text": "GVL, Heating, AKS, Plants, ObjectName, Description"'}
	{attribute 'Tags' := '"LCID": "1033", "Text": "GVL, Heating, DPAD, Plants, ObjectName, Description"'}
	{attribute 'Description' := '"LCID": "1031", "Text": "Anlagenkennzeichnungssystem, Heizsystem Labels Kompensation"'}
	{attribute 'Description' := '"LCID": "1033", "Text": "Data Point Addressing Description, Heating system labels compensation"'}
{endregion}

{attribute 'qualified_only'}
VAR_GLOBAL
	H_HtgCir_Sp_NgtOffs						:FB_BA_Label	:= LblControl_OffsetNightSetpoint;
	H_HtgCir_Sp_SpFlWT						:FB_BA_Label	:= LblFunctions_Setpoint;
	H_HtgCir_Sp_HtgCrv						:FB_BA_Label	:= LblControl_HeatingCurve;
	H_OpMod_OpModMan						:FB_BA_Label	:= LblControl_OperationModeSelection;
	H_OpMod_Sched							:FB_BA_Label	:= LblFunctions_Scheduler;
	H_OpMod_OpModPr							:FB_BA_Label	:= LblControl_PresentOperationMode;
	H_OpMod_Rls								:FB_BA_Label	:= LblFunctions_Enabled;
	
	HtgLmt_Sp								:FB_BA_Label	:= LblFunctions_Setpoint;
	HtgLmt_Q								:FB_BA_Label	:= LblFunctions_OperationalMessage;
	
	
	H_HtgCir_TFl						:FB_BA_Label	:= LblAggregates_TemperatureFlow;
	H_HtgCir_TRt						:FB_BA_Label	:= LblAggregates_TemperatureReturnFlow;
	H_HtgCir_Vlv						:FB_BA_Label	:= LblAggregates_Valve;
	H_HtgCir_Pu							:FB_BA_Label	:= LblAggregates_Pump;
	H_HtgCir_Sp							:FB_BA_Label	:= LblControl_SetpointGeneration;
	H_HtgCir_OpMod						:FB_BA_Label	:= LblControl_OperationMode;
	H_HtgCir_TFlCtrl					:FB_BA_Label	:= LblControl_FlowTemperatureControl;
	H_HtgCir_HtgLmt						:FB_BA_Label	:= LblControl_HeatingLimit;			
END_VAR

// ---- Templates/GVLs/DPAD/Labels/Composition/LblCmpRoomAutomation.TcGVL
{region '#Template'}
	{attribute 'Version' := '1.0.0.0'}
	{attribute 'Tags' := '"LCID": "1031", "Text": "GVL, Room automation, AKS, Plants, ObjectName, Description"'}
	{attribute 'Tags' := '"LCID": "1033", "Text": "GVL, Room automation, DPAD, Plants, ObjectName, Description"'}
	{attribute 'Description' := '"LCID": "1031", "Text": "Anlagenkennzeichnungssystem, Raum Automation Labels Kompensation"'}
	{attribute 'Description' := '"LCID": "1033", "Text": "Data Point Addressing Description, Room automation labels compensation"'}
{endregion}

{attribute 'qualified_only'}
VAR_GLOBAL
	BuildingEnergyLevel_EnergLvlMan					: FB_BA_Label := LblControl_BuildingEnergyLevelManual;
	BuildingEnergyLevel_EnergLvlPr					: FB_BA_Label := LblControl_BuildingEnergyLevelActual;
	BuildingEnergyLevel_Sched						: FB_BA_Label := LblControl_BuildingEnergyLevelSched;
    
	BuildingSpRmT_SumCpsn							: FB_BA_Label := LblControl_SummerCompensation;
	BuildingSpRmT_WinCpsn							: FB_BA_Label := LblControl_WinterCompensation;
	BuildingSpRmT_PrtcHtg							: FB_BA_Label := LblFunctions_SetpointProtectionHeating;
	BuildingSpRmT_EcoHtg							: FB_BA_Label := LblFunctions_SetpointEconomyHeating;
	BuildingSpRmT_PreCmfHtg							: FB_BA_Label := LblFunctions_SetpointPreComfortHeating;
	BuildingSpRmT_CmfHtg							: FB_BA_Label := LblFunctions_SetpointComfortHeating;
	BuildingSpRmT_PrtcCol							: FB_BA_Label := LblFunctions_SetpointProtectionCooling;
	BuildingSpRmT_EcoCol							: FB_BA_Label := LblFunctions_SetpointEconomyCooling;
	BuildingSpRmT_PreCmfCol							: FB_BA_Label := LblFunctions_SetpointPreComfortCooling;
	BuildingSpRmT_CmfCol							: FB_BA_Label := LblFunctions_SetpointComfortCooling;
	BuildingSpRmT_ShiftHtg							: FB_BA_Label := LblControl_SetpointShiftHeating;
	BuildingSpRmT_ShiftCol							: FB_BA_Label := LblControl_SetpointShiftCooling;
	
	BuildingSunprotection_SpIce						: FB_BA_Label := LblControl_SetpointIce;
	BuildingSunprotection_SunPrtcPosIntval			: FB_BA_Label := LblControl_SunProtectionInterval;
	BuildingSunprotection_DeiceTi					: FB_BA_Label := LblControl_DeiceTime;
	BuildingSunprotection_GlobalThAutoValOn			: FB_BA_Label := LblControl_GlobalThermoAutomaticValueOn;
	BuildingSunprotection_GlobalThAutoValOff		: FB_BA_Label := LblControl_GlobalThermoAutomaticValueOff;
	BuildingSunprotection_GlobalTwiLgtAutoValOn		: FB_BA_Label := LblControl_GlobalTwilightAutomaticValueOn;
	BuildingSunprotection_GlobalTwiLgtAutoValOff	: FB_BA_Label := LblControl_GlobalTwilightAutomaticValueOff;
	BuildingSunprotection_IceAlert					: FB_BA_Label := LblControl_IceAlert;
	BuildingSunprotection_GlobalThAutoRlse			: FB_BA_Label := LblControl_GlobalThermoAutomaticRelease;
	BuildingSunprotection_GlobalTwiLgtAutoRlse		: FB_BA_Label := LblControl_GlobalTwilightAutomaticRelease;
	BuildingSunprotection_GlobalResetManMode		: FB_BA_Label := LblControl_GlobalResetManMode;
	
	Facade_DlyStrmOn								: FB_BA_Label := LblControl_TimeDelayStormOn;
	Facade_DlyStrmOff								: FB_BA_Label := LblControl_TimeDelayStormOff;
	Facade_MntnEn									: FB_BA_Label := LblControl_MaintenanceEnable;                    		
	Facade_MntnPos									: FB_BA_Label := LblControl_MaintenancePosition;
	Facade_MntnAngl									: FB_BA_Label := LblControl_MaintenanceAngle;
	Facade_FcdThAutoEn								: FB_BA_Label := LblControl_FacadeThermoAutomaticEnable;
	Facade_FcdThAutoColPos							: FB_BA_Label := LblControl_FacadeThermoAutomaticCoolingPosition;
	Facade_FcdThAutoColAngl							: FB_BA_Label := LblControl_FacadeThermoAutomaticCoolingAngle;
	Facade_FcdTwiLgtAutoEn							: FB_BA_Label := LblControl_FacadeTwilightAutomaticEnable;
	Facade_SunPrtcValOn								: FB_BA_Label := LblControl_SunProtectionValueOn;
	Facade_SunPrtcValOff							: FB_BA_Label := LblControl_SunProtectionValueOff;
	Facade_SunPrtcDlyOn								: FB_BA_Label := LblControl_TimeDelaySunProtectionOn;
	Facade_SunPrtcDlyOff							: FB_BA_Label := LblControl_TimeDelaySunProtectionOff;
	Facade_FcdParkEn								: FB_BA_Label := LblControl_FacadeParkingEnable;
	Facade_FcdParkPos								: FB_BA_Label := LblControl_FacadeParkingPosition;
	Facade_FcdParkAngl								: FB_BA_Label := LblControl_FacadeParkingAngle;
	Facade_WndPrtcState								: FB_BA_Label := LblControl_WindProtectionState;
	Facade_SunPrtcState								: FB_BA_Label := LblControl_SunProtectionState;
    
	SunBld_LocInputPos								: FB_BA_Label := LblControl_SetpointSunblindPosition;
	SunBld_LocInputAngl								: FB_BA_Label := LblControl_SetpointSunblindAngle;
	SunBld_LocButtonStart							: FB_BA_Label := LblControl_CommandSunblindStart;
	SunBld_ActlPos									: FB_BA_Label := LblControl_FeedbackSunblindPosition;
	SunBld_ActlAngl									: FB_BA_Label := LblControl_FeedbackSunblindAngle;
	SunBld_ActlPrio									: FB_BA_Label := LblControl_FeedbackSunblindPrio;
	SunBld_ManSwi									: FB_BA_Label := LblControl_ButtonSunblind;
		
	HeatCoolAxisAnlg_RmTSen							: FB_BA_Label := LblAggregates_TemperatureRoomAir;
	HeatCoolAxisAnlg_RmTAdj							: FB_BA_Label := LblAggregates_RoomControlUnit;
	HeatCoolAxisAnlg_PrtcDetc						: FB_BA_Label := LblAggregates_PresenceSwitches;
	HeatCoolAxisAnlg_WdwCon							: FB_BA_Label := LblAggregates_WindowContact;
	HeatCoolAxisAnlg_VlvHtg							: FB_BA_Label :=(sObjName:='VEN',sDescr:='Heizventil');
 	HeatCoolAxisAnlg_VlvCol							: FB_BA_Label :=(sObjName:='VEN',sDescr:='Kuehlventil');
 	HeatCoolAxisAnlg_Ctrl							: FB_BA_Label := LblControl_RoomTemperatureControl;
 	HeatCoolAxisAnlg_Ctrl_CtrlHtg					: FB_BA_Label :=(sObjName:='LPH',sDescr:='Heizregler');
 	HeatCoolAxisAnlg_Ctrl_CtrlCol					: FB_BA_Label :=(sObjName:='LPC',sDescr:='Kuehlregler');
	HeatCoolAxisAnlg_DewPoint						: FB_BA_Label := LblAggregates_MonitorDewPoint;

	SunBldZone_SunBld								: FB_BA_Label := LblAggregates_Blind;
                                          	
//	RoomAutomation_RoomGeneral						: FB_BA_Label := LabelPlants.Room_automation;
	
	RoomGeneral_FcdEast								: FB_BA_Label := LblControl_Facade;
END_VAR

// ---- Templates/GVLs/DPAD/Labels/Composition/LblUniControl.TcGVL
{region '#Template'}
	{attribute 'Version' := '1.0.0.0'}
	{attribute 'Tags' := '"LCID": "1031", "Text": "GVL, Universal, AKS, Plants, ObjectName, Description"'}
	{attribute 'Tags' := '"LCID": "1033", "Text": "GVL, Universal, DPAD, Plants, ObjectName, Description"'}
	{attribute 'Description' := '"LCID": "1031", "Text": "Anlagenkennzeichnungssystem, Universal Labels Kompensation"'}
	{attribute 'Description' := '"LCID": "1033", "Text": "Data Point Addressing Description, Universal labels compensation"'}
{endregion}

